REGION Network 2: Drive control B nok
   RUNG wire#powerrail
      Contact( "Servo Control"."B"."drive error" )
      wire#w1
      Coil( "Faults&warnings"."Status Nok"."Drive controller B NK" )
   END_RUNG
   RUNG wire#powerrail
      Contact( "Servo Control"."B"."Communication Error" )
   END_RUNG wire#w1
   RUNG wire#powerrail
      I_Contact( "Alarm Drive 2" )
   END_RUNG wire#w1
   RUNG wire#w1
      Coil( "Alarm_DB".input.alarm[10] )
   END_RUNG
   // the same network as SCL:
   "Faults&warnings"."Status Nok"."Drive controller B NK" := "Servo Control"."B"."drive error" OR "Servo Control"."B"."Communication Error" OR NOT "Alarm Drive 2";
   "Alarm_DB".input.alarm[10] := "Faults&warnings"."Status Nok"."Drive controller B NK";
END_REGION

REGION Network 3: Agitator A Fault
   RUNG wire#powerrail
      Contact( "A4-Agitator A1 fault" )
      Coil( "Faults&warnings"."Status Nok"."Agitator A Fault" )
   END_RUNG
   // the same network as SCL:
   "Faults&warnings"."Status Nok"."Agitator A Fault" := "A4-Agitator A1 fault";
END_REGION

REGION Network 4: Agitator B Fault
   RUNG wire#powerrail
      Contact( "A5-Agitator A2 fault" )
      Coil( "Faults&warnings"."Status Nok"."Agitator B Fault" )
   END_RUNG
   // the same network as SCL:
   "Faults&warnings"."Status Nok"."Agitator B Fault" := "A5-Agitator A2 fault";
END_REGION

REGION Network 5: pressure sensor Pump A inlet
   RUNG wire#powerrail
      { S7_Templates := "SrcType := Int" } GE_Contact(in1 := "Pressure sensor Pump Inlet A", in2 := 32767)
      { S7_Templates := "SrcType := Int" } EQ_Contact(in1 := "Control".Pressure_sensor_select, in2 := 0)
      wire#w1
      Coil( "Faults&warnings"."Status Nok"."Pressure sensor Pump A Inlet" )
   END_RUNG
   RUNG wire#powerrail
      { S7_Templates := "SrcType := Int" } GE_Contact(in1 := "Pressure sensor Pump Inlet A_mA", in2 := 32767)
      { S7_Templates := "SrcType := Int" } EQ_Contact(in1 := "Control".Pressure_sensor_select, in2 := 1)
   END_RUNG wire#w1
   // the same network as SCL:
   "Faults&warnings"."Status Nok"."Pressure sensor Pump A Inlet" := (("Pressure sensor Pump Inlet A" >= 32767) AND ("Control".Pressure_sensor_select = 0)) OR (("Pressure sensor Pump Inlet A_mA" >= 32767) AND ("Control".Pressure_sensor_select = 1));
END_REGION

REGION Network 6: pressure sensor Pump A outlet
   RUNG wire#powerrail
      { S7_Templates := "SrcType := Int" } GE_Contact(in1 := "Pressure Sensor Pump Outlet A", in2 := 32767)
      I_Contact( "AlwaysFALSE" )
      Contact( "pressure".Outlet_PT_ENABLE )
      wire#w1
      Coil( "Faults&warnings"."Status Nok"."Pressure sensor Pump A Outlet" )
   END_RUNG
   RUNG wire#w1
      Coil( "Alarm_DB".input.alarm[81] )
   END_RUNG
   // the same network as SCL:
   "Faults&warnings"."Status Nok"."Pressure sensor Pump A Outlet" := ("Pressure Sensor Pump Outlet A" >= 32767) AND NOT "AlwaysFALSE" AND "pressure".Outlet_PT_ENABLE;
   "Alarm_DB".input.alarm[81] := "Faults&warnings"."Status Nok"."Pressure sensor Pump A Outlet";
END_REGION

REGION Network 7: pressure sensor Pump B inlet
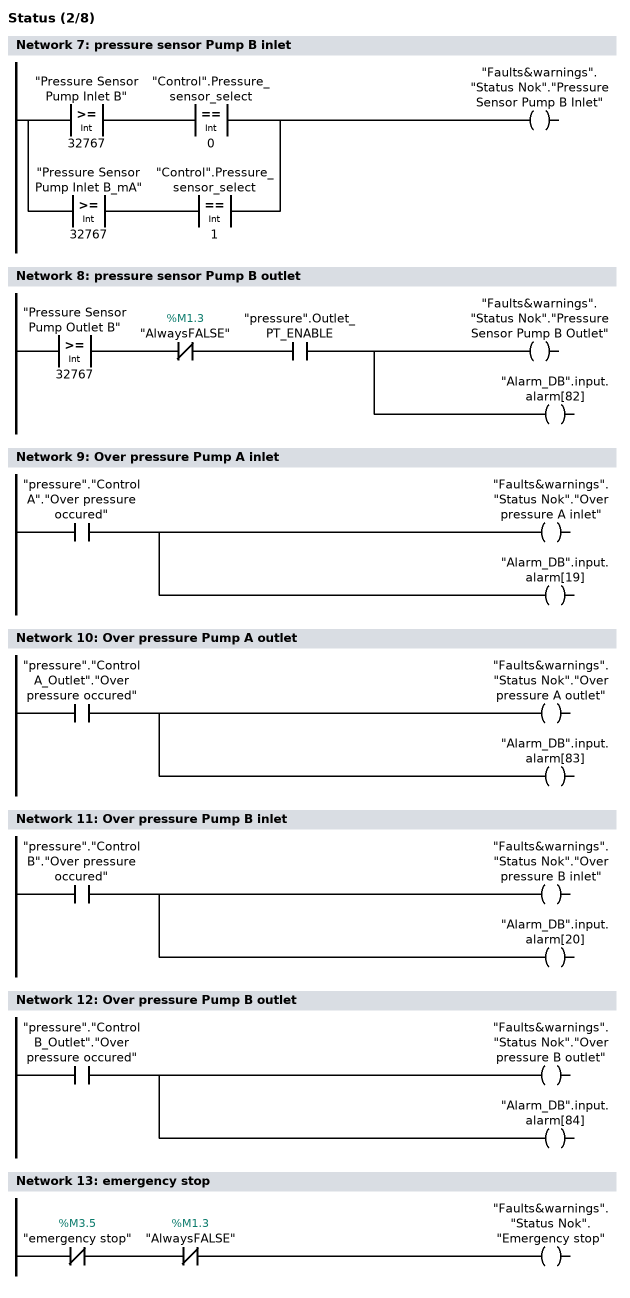
   RUNG wire#powerrail
      { S7_Templates := "SrcType := Int" } GE_Contact(in1 := "Pressure Sensor Pump Inlet B", in2 := 32767)
      { S7_Templates := "SrcType := Int" } EQ_Contact(in1 := "Control".Pressure_sensor_select, in2 := 0)
      wire#w1
      Coil( "Faults&warnings"."Status Nok"."Pressure Sensor Pump B Inlet" )
   END_RUNG
   RUNG wire#powerrail
      { S7_Templates := "SrcType := Int" } GE_Contact(in1 := "Pressure Sensor Pump Inlet B_mA", in2 := 32767)
      { S7_Templates := "SrcType := Int" } EQ_Contact(in1 := "Control".Pressure_sensor_select, in2 := 1)
   END_RUNG wire#w1
   // the same network as SCL:
   "Faults&warnings"."Status Nok"."Pressure Sensor Pump B Inlet" := (("Pressure Sensor Pump Inlet B" >= 32767) AND ("Control".Pressure_sensor_select = 0)) OR (("Pressure Sensor Pump Inlet B_mA" >= 32767) AND ("Control".Pressure_sensor_select = 1));
END_REGION

REGION Network 8: pressure sensor Pump B outlet
   RUNG wire#powerrail
      { S7_Templates := "SrcType := Int" } GE_Contact(in1 := "Pressure Sensor Pump Outlet B", in2 := 32767)
      I_Contact( "AlwaysFALSE" )
      Contact( "pressure".Outlet_PT_ENABLE )
      wire#w1
      Coil( "Faults&warnings"."Status Nok"."Pressure Sensor Pump B Outlet" )
   END_RUNG
   RUNG wire#w1
      Coil( "Alarm_DB".input.alarm[82] )
   END_RUNG
   // the same network as SCL:
   "Faults&warnings"."Status Nok"."Pressure Sensor Pump B Outlet" := ("Pressure Sensor Pump Outlet B" >= 32767) AND NOT "AlwaysFALSE" AND "pressure".Outlet_PT_ENABLE;
   "Alarm_DB".input.alarm[82] := "Faults&warnings"."Status Nok"."Pressure Sensor Pump B Outlet";
END_REGION

REGION Network 9: Over pressure Pump A inlet
   RUNG wire#powerrail
      Contact( "pressure"."Control A"."Over pressure occured" )
      wire#w1
      Coil( "Faults&warnings"."Status Nok"."Over pressure A inlet" )
   END_RUNG
   RUNG wire#w1
      Coil( "Alarm_DB".input.alarm[19] )
   END_RUNG
   // the same network as SCL:
   "Faults&warnings"."Status Nok"."Over pressure A inlet" := "pressure"."Control A"."Over pressure occured";
   "Alarm_DB".input.alarm[19] := "pressure"."Control A"."Over pressure occured";
END_REGION

REGION Network 10: Over pressure Pump A outlet
   RUNG wire#powerrail
      Contact( "pressure"."Control A_Outlet"."Over pressure occured" )
      wire#w1
      Coil( "Faults&warnings"."Status Nok"."Over pressure A outlet" )
   END_RUNG
   RUNG wire#w1
      Coil( "Alarm_DB".input.alarm[83] )
   END_RUNG
   // the same network as SCL:
   "Faults&warnings"."Status Nok"."Over pressure A outlet" := "pressure"."Control A_Outlet"."Over pressure occured";
   "Alarm_DB".input.alarm[83] := "pressure"."Control A_Outlet"."Over pressure occured";
END_REGION

REGION Network 11: Over pressure Pump B inlet
   RUNG wire#powerrail
      Contact( "pressure"."Control B"."Over pressure occured" )
      wire#w1
      Coil( "Faults&warnings"."Status Nok"."Over pressure B inlet" )
   END_RUNG
   RUNG wire#w1
      Coil( "Alarm_DB".input.alarm[20] )
   END_RUNG
   // the same network as SCL:
   "Faults&warnings"."Status Nok"."Over pressure B inlet" := "pressure"."Control B"."Over pressure occured";
   "Alarm_DB".input.alarm[20] := "pressure"."Control B"."Over pressure occured";
END_REGION

REGION Network 12: Over pressure Pump B outlet
   RUNG wire#powerrail
      Contact( "pressure"."Control B_Outlet"."Over pressure occured" )
      wire#w1
      Coil( "Faults&warnings"."Status Nok"."Over pressure B outlet" )
   END_RUNG
   RUNG wire#w1
      Coil( "Alarm_DB".input.alarm[84] )
   END_RUNG
   // the same network as SCL:
   "Faults&warnings"."Status Nok"."Over pressure B outlet" := "pressure"."Control B_Outlet"."Over pressure occured";
   "Alarm_DB".input.alarm[84] := "pressure"."Control B_Outlet"."Over pressure occured";
END_REGION

REGION Network 13: emergency stop
   RUNG wire#powerrail
      I_Contact( "emergency stop" )
      I_Contact( "AlwaysFALSE" )
      Coil( "Faults&warnings"."Status Nok"."Emergency stop" )
   END_RUNG
   // the same network as SCL:
   "Faults&warnings"."Status Nok"."Emergency stop" := NOT "emergency stop" AND NOT "AlwaysFALSE";
END_REGION

REGION Network 14: HEATER OK
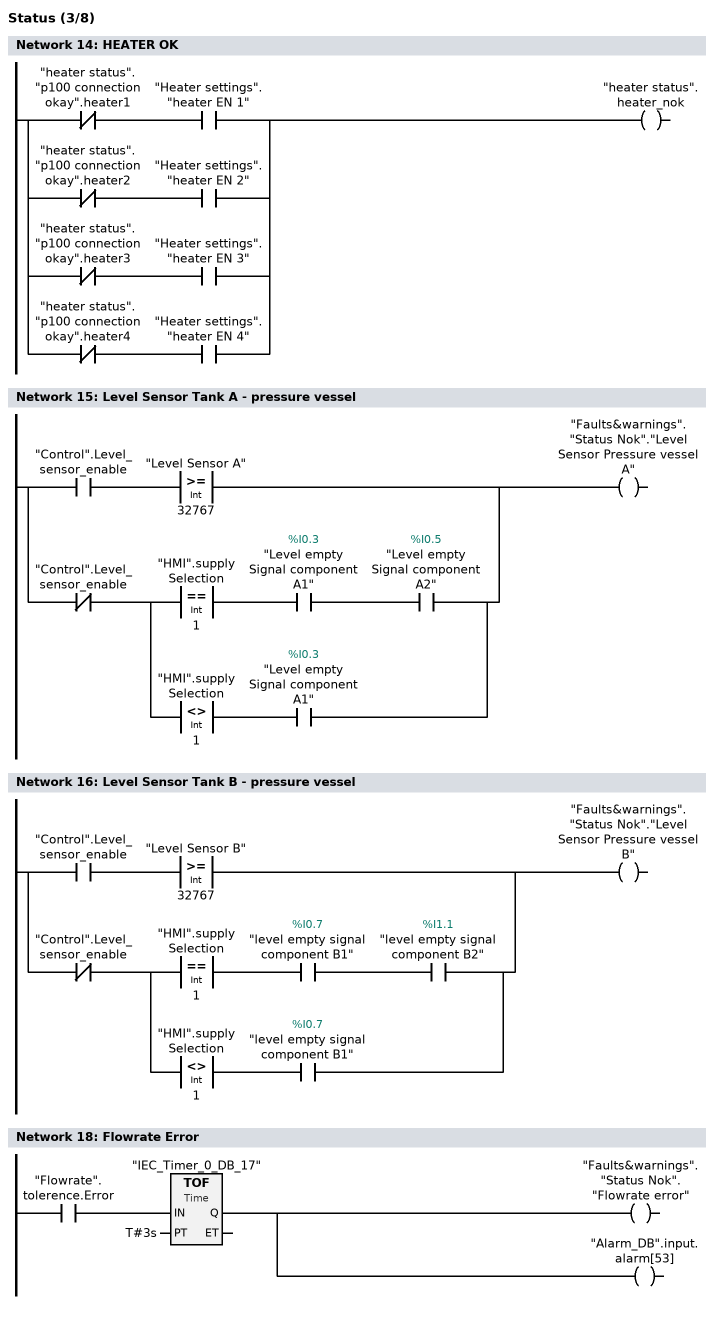
   RUNG wire#powerrail
      I_Contact( "heater status"."p100 connection okay".heater1 )
      Contact( "Heater settings"."heater EN 1" )
      wire#w1
      Coil( "heater status".heater_nok )
   END_RUNG
   RUNG wire#powerrail
      I_Contact( "heater status"."p100 connection okay".heater2 )
      Contact( "Heater settings"."heater EN 2" )
   END_RUNG wire#w1
   RUNG wire#powerrail
      I_Contact( "heater status"."p100 connection okay".heater3 )
      Contact( "Heater settings"."heater EN 3" )
   END_RUNG wire#w1
   RUNG wire#powerrail
      I_Contact( "heater status"."p100 connection okay".heater4 )
      Contact( "Heater settings"."heater EN 4" )
   END_RUNG wire#w1
   // the same network as SCL:
   "heater status".heater_nok := (NOT "heater status"."p100 connection okay".heater1 AND "Heater settings"."heater EN 1") OR (NOT "heater status"."p100 connection okay".heater2 AND "Heater settings"."heater EN 2") OR (NOT "heater status"."p100 connection okay".heater3 AND "Heater settings"."heater EN 3") OR (NOT "heater status"."p100 connection okay".heater4 AND "Heater settings"."heater EN 4");
END_REGION

REGION Network 15: Level Sensor Tank A - pressure vessel
   RUNG wire#powerrail
      Contact( "Control".Level_sensor_enable )
      { S7_Templates := "SrcType := Int" } GE_Contact(in1 := "Level Sensor A", in2 := 32767)
      wire#w1
      Coil( "Faults&warnings"."Status Nok"."Level Sensor Pressure vessel A" )
   END_RUNG
   RUNG wire#powerrail
      I_Contact( "Control".Level_sensor_enable )
      wire#w2
      { S7_Templates := "SrcType := Int" } EQ_Contact(in1 := "HMI".supplySelection, in2 := 1)
      Contact( "Level empty Signal component A1" )
      Contact( "Level empty Signal component A2" )
   END_RUNG wire#w1
   RUNG wire#w2
      { S7_Templates := "SrcType := Int" } NE_Contact(in1 := "HMI".supplySelection, in2 := 1)
      Contact( "Level empty Signal component A1" )
   END_RUNG wire#w1
   // the same network as SCL:
   "Faults&warnings"."Status Nok"."Level Sensor Pressure vessel A" := ("Control".Level_sensor_enable AND ("Level Sensor A" >= 32767)) OR (NOT "Control".Level_sensor_enable AND ((("HMI".supplySelection = 1) AND "Level empty Signal component A1" AND "Level empty Signal component A2") OR (("HMI".supplySelection <> 1) AND "Level empty Signal component A1")));
END_REGION

REGION Network 16: Level Sensor Tank B - pressure vessel
   RUNG wire#powerrail
      Contact( "Control".Level_sensor_enable )
      { S7_Templates := "SrcType := Int" } GE_Contact(in1 := "Level Sensor B", in2 := 32767)
      wire#w1
      Coil( "Faults&warnings"."Status Nok"."Level Sensor Pressure vessel B" )
   END_RUNG
   RUNG wire#powerrail
      I_Contact( "Control".Level_sensor_enable )
      wire#w2
      { S7_Templates := "SrcType := Int" } EQ_Contact(in1 := "HMI".supplySelection, in2 := 1)
      Contact( "level empty signal component B1" )
      Contact( "level empty signal component B2" )
   END_RUNG wire#w1
   RUNG wire#w2
      { S7_Templates := "SrcType := Int" } NE_Contact(in1 := "HMI".supplySelection, in2 := 1)
      Contact( "level empty signal component B1" )
   END_RUNG wire#w1
   // the same network as SCL:
   "Faults&warnings"."Status Nok"."Level Sensor Pressure vessel B" := ("Control".Level_sensor_enable AND ("Level Sensor B" >= 32767)) OR (NOT "Control".Level_sensor_enable AND ((("HMI".supplySelection = 1) AND "level empty signal component B1" AND "level empty signal component B2") OR (("HMI".supplySelection <> 1) AND "level empty signal component B1")));
END_REGION

REGION Network 17 (SCL): low level and empty level non tandum
   "Alarm_DB".input.alarm[40] := "Faults&warnings"."Status Nok"."Low level A1"  := "level"."Low level occured A";
   "Alarm_DB".input.alarm[42] := "Faults&warnings"."Status Nok"."Low level B1" := "level"."Low level occured B";

   "Faults&warnings"."Status Nok"."Level empty A1" := "level"."Level Empty A";
   "Alarm_DB".input.alarm[21] := "Faults&warnings"."Status Nok"."Level empty A1" OR "Temp".bit20;
   "Faults&warnings"."Status Nok"."Level empty B1" := "level"."Level Empty B";
   "Alarm_DB".input.alarm[23] := "Faults&warnings"."Status Nok"."Level empty B1" OR "Temp".bit21;

   "Faults&warnings"."Status Nok"."Level Low Drum A1" := "level"."Drum Level Low A1" AND "HMI".supplySelection = 1;
   "Faults&warnings"."Status Nok"."Level Low Drum A2" := "level"."Drum Level Low A2" AND "HMI".supplySelection = 1;
   "Faults&warnings"."Status Nok"."Level Low Drum B1" := "level"."Drum Level Low B1" AND "HMI".supplySelection = 1;
   "Faults&warnings"."Status Nok"."Level Low Drum B2" := "level"."Drum Level Low B2" AND "HMI".supplySelection = 1;

   "Faults&warnings"."Status Nok"."Level Empty Drum A1" := "level"."Drum Level Empty A1" AND "HMI".supplySelection = 1;
   "Faults&warnings"."Status Nok"."Level Empty Drum A2" := "level"."Drum Level Empty A2" AND "HMI".supplySelection = 1;
   "Faults&warnings"."Status Nok"."Level Empty Drum B1" := "level"."Drum Level Empty B1" AND "HMI".supplySelection = 1;
   "Faults&warnings"."Status Nok"."Level Empty Drum B2" := "level"."Drum Level Empty B2" AND "HMI".supplySelection = 1;
END_REGION

REGION Network 18: Flowrate Error
   RUNG wire#powerrail
      Contact( "Flowrate".tolerence.Error )
      { S7_Templates := "time_type := Time" } "IEC_Timer_0_DB_17".TOF(pt := T#3s, et =>)
      wire#w1
      Coil( "Faults&warnings"."Status Nok"."Flowrate error" )
   END_RUNG
   RUNG wire#w1
      Coil( "Alarm_DB".input.alarm[53] )
   END_RUNG
   // the same network as SCL:
   "IEC_Timer_0_DB_17".TOF(IN := "Flowrate".tolerence.Error, PT := T#3s);
   "Faults&warnings"."Status Nok"."Flowrate error" := "IEC_Timer_0_DB_17".Q;
   "Alarm_DB".input.alarm[53] := "IEC_Timer_0_DB_17".Q;
END_REGION

REGION Network 19: Critical Fault stop A metering
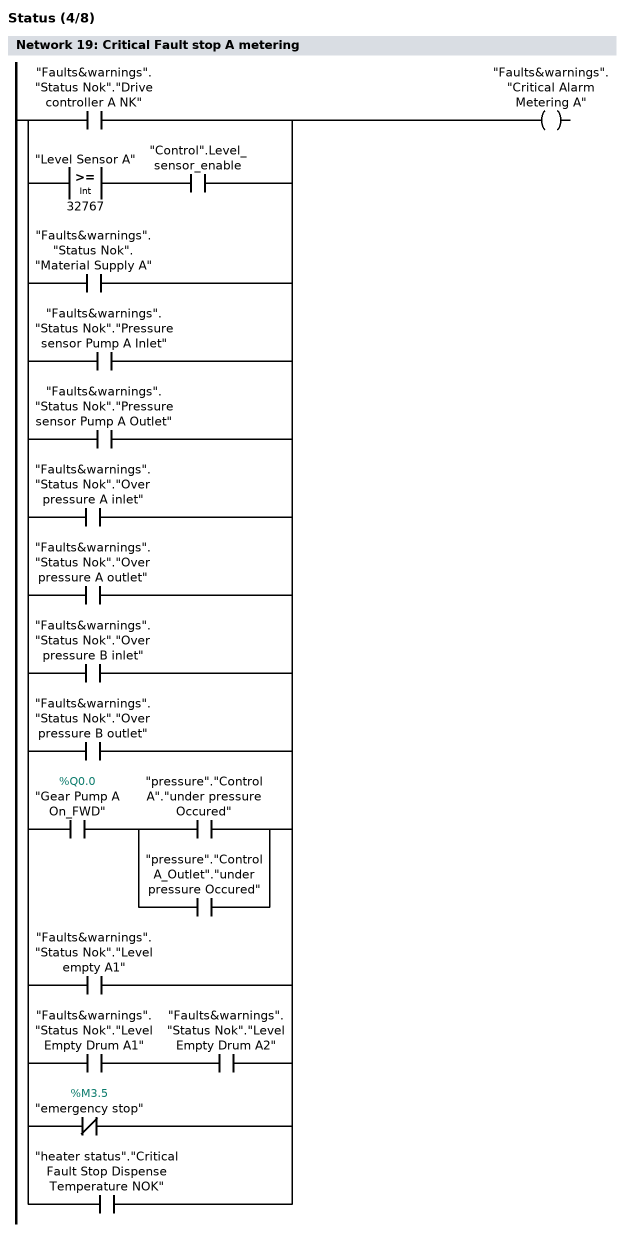
   RUNG wire#powerrail
      Contact( "Faults&warnings"."Status Nok"."Drive controller A NK" )
      wire#w1
      Coil( "Faults&warnings"."Critical Alarm Metering A" )
   END_RUNG
   RUNG wire#powerrail
      { S7_Templates := "SrcType := Int" } GE_Contact(in1 := "Level Sensor A", in2 := 32767)
      Contact( "Control".Level_sensor_enable )
   END_RUNG wire#w1
   RUNG wire#powerrail
      Contact( "Faults&warnings"."Status Nok"."Material Supply A" )
   END_RUNG wire#w1
   RUNG wire#powerrail
      Contact( "Faults&warnings"."Status Nok"."Pressure sensor Pump A Inlet" )
   END_RUNG wire#w1
   RUNG wire#powerrail
      Contact( "Faults&warnings"."Status Nok"."Pressure sensor Pump A Outlet" )
   END_RUNG wire#w1
   RUNG wire#powerrail
      Contact( "Faults&warnings"."Status Nok"."Over pressure A inlet" )
   END_RUNG wire#w1
   RUNG wire#powerrail
      Contact( "Faults&warnings"."Status Nok"."Over pressure A outlet" )
   END_RUNG wire#w1
   RUNG wire#powerrail
      Contact( "Faults&warnings"."Status Nok"."Over pressure B inlet" )
   END_RUNG wire#w1
   RUNG wire#powerrail
      Contact( "Faults&warnings"."Status Nok"."Over pressure B outlet" )
   END_RUNG wire#w1
   RUNG wire#powerrail
      Contact( "Gear Pump A On_FWD" )
      wire#w2
      Contact( "pressure"."Control A"."under pressure Occured" )
   END_RUNG wire#w1
   RUNG wire#w2
      Contact( "pressure"."Control A_Outlet"."under pressure Occured" )
   END_RUNG wire#w1
   RUNG wire#powerrail
      Contact( "Faults&warnings"."Status Nok"."Level empty A1" )
   END_RUNG wire#w1
   RUNG wire#powerrail
      Contact( "Faults&warnings"."Status Nok"."Level Empty Drum A1" )
      Contact( "Faults&warnings"."Status Nok"."Level Empty Drum A2" )
   END_RUNG wire#w1
   RUNG wire#powerrail
      I_Contact( "emergency stop" )
   END_RUNG wire#w1
   RUNG wire#powerrail
      Contact( "heater status"."Critical Fault Stop Dispense Temperature NOK" )
   END_RUNG wire#w1
   // the same network as SCL:
   "Faults&warnings"."Critical Alarm Metering A" := "Faults&warnings"."Status Nok"."Drive controller A NK" OR (("Level Sensor A" >= 32767) AND "Control".Level_sensor_enable) OR "Faults&warnings"."Status Nok"."Material Supply A" OR "Faults&warnings"."Status Nok"."Pressure sensor Pump A Inlet" OR "Faults&warnings"."Status Nok"."Pressure sensor Pump A Outlet" OR "Faults&warnings"."Status Nok"."Over pressure A inlet" OR "Faults&warnings"."Status Nok"."Over pressure A outlet" OR "Faults&warnings"."Status Nok"."Over pressure B inlet" OR "Faults&warnings"."Status Nok"."Over pressure B outlet" OR ("Gear Pump A On_FWD" AND ("pressure"."Control A"."under pressure Occured" OR "pressure"."Control A_Outlet"."under pressure Occured")) OR "Faults&warnings"."Status Nok"."Level empty A1" OR ("Faults&warnings"."Status Nok"."Level Empty Drum A1" AND "Faults&warnings"."Status Nok"."Level Empty Drum A2") OR NOT "emergency stop" OR "heater status"."Critical Fault Stop Dispense Temperature NOK";
END_REGION

REGION Network 20: Critical Fault stop B metering
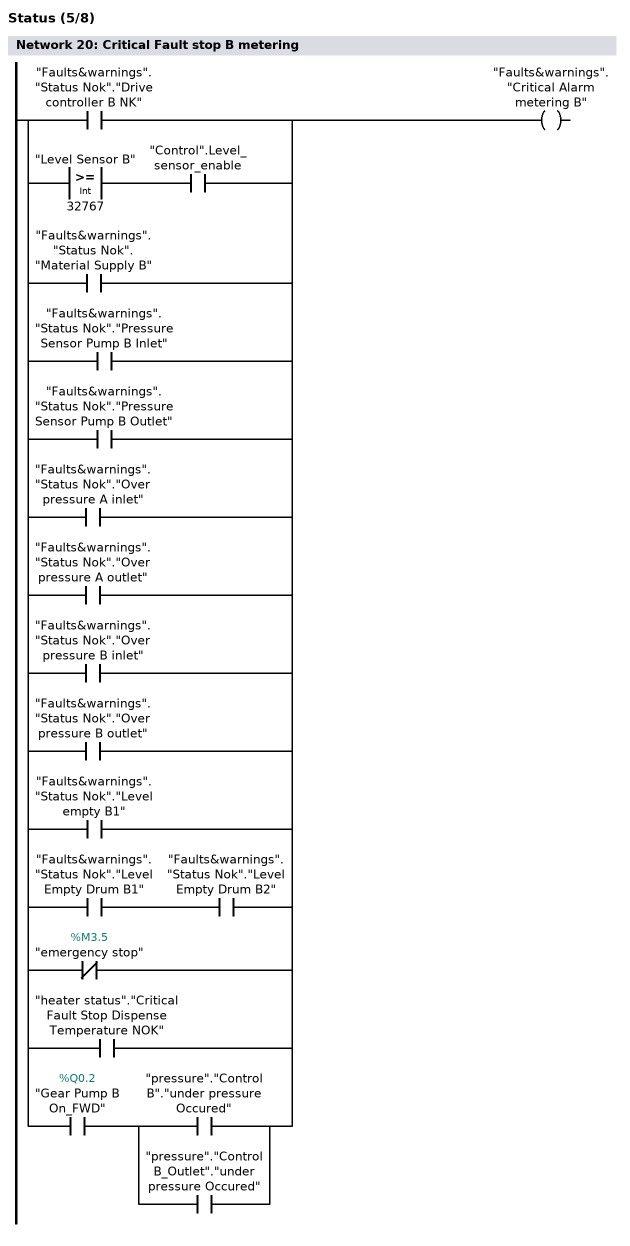
   RUNG wire#powerrail
      Contact( "Faults&warnings"."Status Nok"."Drive controller B NK" )
      wire#w1
      Coil( "Faults&warnings"."Critical Alarm metering B" )
   END_RUNG
   RUNG wire#powerrail
      { S7_Templates := "SrcType := Int" } GE_Contact(in1 := "Level Sensor B", in2 := 32767)
      Contact( "Control".Level_sensor_enable )
   END_RUNG wire#w1
   RUNG wire#powerrail
      Contact( "Faults&warnings"."Status Nok"."Material Supply B" )
   END_RUNG wire#w1
   RUNG wire#powerrail
      Contact( "Faults&warnings"."Status Nok"."Pressure Sensor Pump B Inlet" )
   END_RUNG wire#w1
   RUNG wire#powerrail
      Contact( "Faults&warnings"."Status Nok"."Pressure Sensor Pump B Outlet" )
   END_RUNG wire#w1
   RUNG wire#powerrail
      Contact( "Faults&warnings"."Status Nok"."Over pressure A inlet" )
   END_RUNG wire#w1
   RUNG wire#powerrail
      Contact( "Faults&warnings"."Status Nok"."Over pressure A outlet" )
   END_RUNG wire#w1
   RUNG wire#powerrail
      Contact( "Faults&warnings"."Status Nok"."Over pressure B inlet" )
   END_RUNG wire#w1
   RUNG wire#powerrail
      Contact( "Faults&warnings"."Status Nok"."Over pressure B outlet" )
   END_RUNG wire#w1
   RUNG wire#powerrail
      Contact( "Faults&warnings"."Status Nok"."Level empty B1" )
   END_RUNG wire#w1
   RUNG wire#powerrail
      Contact( "Faults&warnings"."Status Nok"."Level Empty Drum B1" )
      Contact( "Faults&warnings"."Status Nok"."Level Empty Drum B2" )
   END_RUNG wire#w1
   RUNG wire#powerrail
      I_Contact( "emergency stop" )
   END_RUNG wire#w1
   RUNG wire#powerrail
      Contact( "heater status"."Critical Fault Stop Dispense Temperature NOK" )
   END_RUNG wire#w1
   RUNG wire#powerrail
      Contact( "Gear Pump B On_FWD" )
      wire#w2
      Contact( "pressure"."Control B"."under pressure Occured" )
   END_RUNG wire#w1
   RUNG wire#w2
      Contact( "pressure"."Control B_Outlet"."under pressure Occured" )
   END_RUNG wire#w1
   // the same network as SCL:
   "Faults&warnings"."Critical Alarm metering B" := "Faults&warnings"."Status Nok"."Drive controller B NK" OR (("Level Sensor B" >= 32767) AND "Control".Level_sensor_enable) OR "Faults&warnings"."Status Nok"."Material Supply B" OR "Faults&warnings"."Status Nok"."Pressure Sensor Pump B Inlet" OR "Faults&warnings"."Status Nok"."Pressure Sensor Pump B Outlet" OR "Faults&warnings"."Status Nok"."Over pressure A inlet" OR "Faults&warnings"."Status Nok"."Over pressure A outlet" OR "Faults&warnings"."Status Nok"."Over pressure B inlet" OR "Faults&warnings"."Status Nok"."Over pressure B outlet" OR "Faults&warnings"."Status Nok"."Level empty B1" OR ("Faults&warnings"."Status Nok"."Level Empty Drum B1" AND "Faults&warnings"."Status Nok"."Level Empty Drum B2") OR NOT "emergency stop" OR "heater status"."Critical Fault Stop Dispense Temperature NOK" OR ("Gear Pump B On_FWD" AND ("pressure"."Control B"."under pressure Occured" OR "pressure"."Control B_Outlet"."under pressure Occured"));
END_REGION

REGION Network 21: critical alarm AB
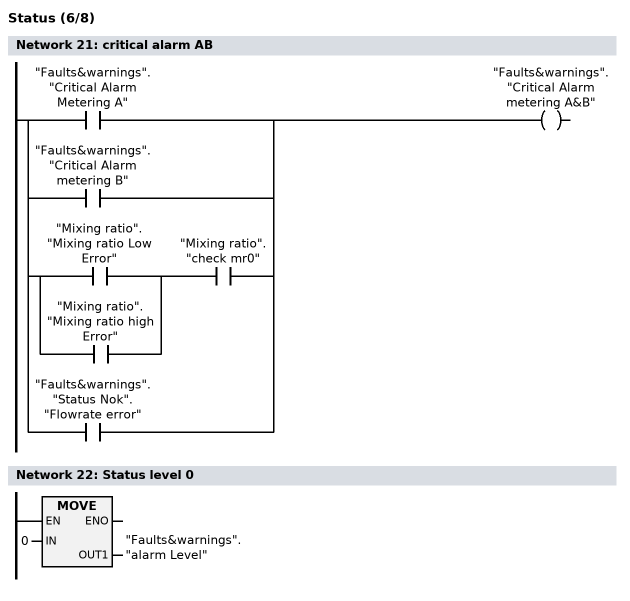
   RUNG wire#powerrail
      Contact( "Faults&warnings"."Critical Alarm Metering A" )
      wire#w1
      Coil( "Faults&warnings"."Critical Alarm metering A&B" )
   END_RUNG
   RUNG wire#powerrail
      Contact( "Faults&warnings"."Critical Alarm metering B" )
   END_RUNG wire#w1
   RUNG wire#powerrail
      Contact( "Mixing ratio"."Mixing ratio Low  Error" )
      wire#w2
      Contact( "Mixing ratio"."check mr0" )
   END_RUNG wire#w1
   RUNG wire#powerrail
      Contact( "Mixing ratio"."Mixing ratio high Error" )
   END_RUNG wire#w2
   RUNG wire#powerrail
      Contact( "Faults&warnings"."Status Nok"."Flowrate error" )
   END_RUNG wire#w1
   // the same network as SCL:
   "Faults&warnings"."Critical Alarm metering A&B" := "Faults&warnings"."Critical Alarm Metering A" OR "Faults&warnings"."Critical Alarm metering B" OR (("Mixing ratio"."Mixing ratio Low  Error" OR "Mixing ratio"."Mixing ratio high Error") AND "Mixing ratio"."check mr0") OR "Faults&warnings"."Status Nok"."Flowrate error";
END_REGION

REGION Network 22: Status level 0
   RUNG wire#powerrail
      Move(in := 0, out1 => "Faults&warnings"."alarm Level")
   END_RUNG
   // the same network as SCL:
   "Faults&warnings"."alarm Level" := 0;
END_REGION

REGION Network 23: Status level 1/warning
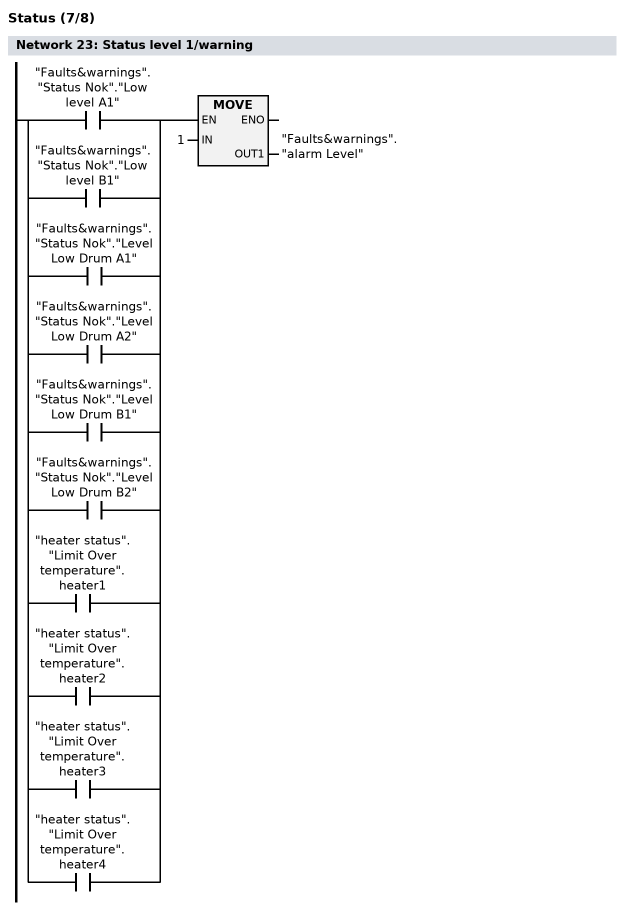
   RUNG wire#powerrail
      Contact( "Faults&warnings"."Status Nok"."Low level A1" )
      wire#w1
      Move(in := 1, out1 => "Faults&warnings"."alarm Level")
   END_RUNG
   RUNG wire#powerrail
      Contact( "Faults&warnings"."Status Nok"."Low level B1" )
   END_RUNG wire#w1
   RUNG wire#powerrail
      Contact( "Faults&warnings"."Status Nok"."Level Low Drum A1" )
   END_RUNG wire#w1
   RUNG wire#powerrail
      Contact( "Faults&warnings"."Status Nok"."Level Low Drum A2" )
   END_RUNG wire#w1
   RUNG wire#powerrail
      Contact( "Faults&warnings"."Status Nok"."Level Low Drum B1" )
   END_RUNG wire#w1
   RUNG wire#powerrail
      Contact( "Faults&warnings"."Status Nok"."Level Low Drum B2" )
   END_RUNG wire#w1
   RUNG wire#powerrail
      Contact( "heater status"."Limit Over temperature".heater1 )
   END_RUNG wire#w1
   RUNG wire#powerrail
      Contact( "heater status"."Limit Over temperature".heater2 )
   END_RUNG wire#w1
   RUNG wire#powerrail
      Contact( "heater status"."Limit Over temperature".heater3 )
   END_RUNG wire#w1
   RUNG wire#powerrail
      Contact( "heater status"."Limit Over temperature".heater4 )
   END_RUNG wire#w1
   // the same network as SCL:
   IF "Faults&warnings"."Status Nok"."Low level A1" OR "Faults&warnings"."Status Nok"."Low level B1" OR "Faults&warnings"."Status Nok"."Level Low Drum A1" OR "Faults&warnings"."Status Nok"."Level Low Drum A2" OR "Faults&warnings"."Status Nok"."Level Low Drum B1" OR "Faults&warnings"."Status Nok"."Level Low Drum B2" OR "heater status"."Limit Over temperature".heater1 OR "heater status"."Limit Over temperature".heater2 OR "heater status"."Limit Over temperature".heater3 OR "heater status"."Limit Over temperature".heater4 THEN
       "Faults&warnings"."alarm Level" := 1;
   END_IF;
END_REGION

REGION Network 24: Status level 1/fault
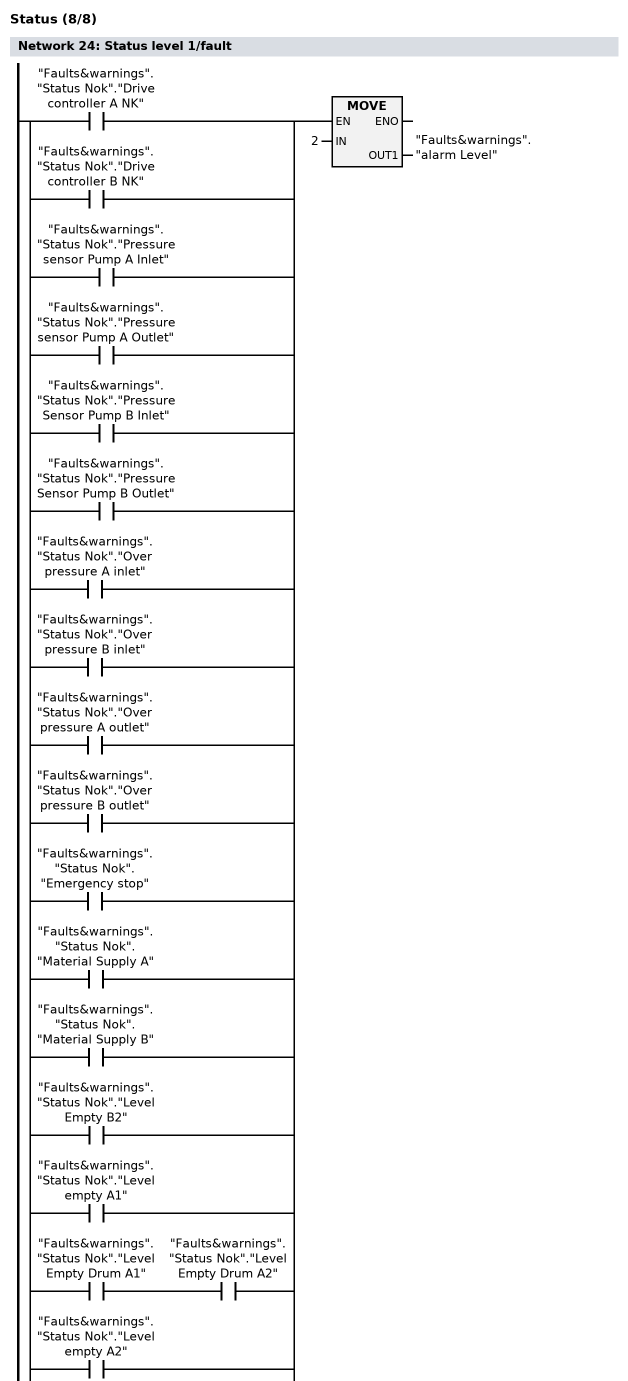
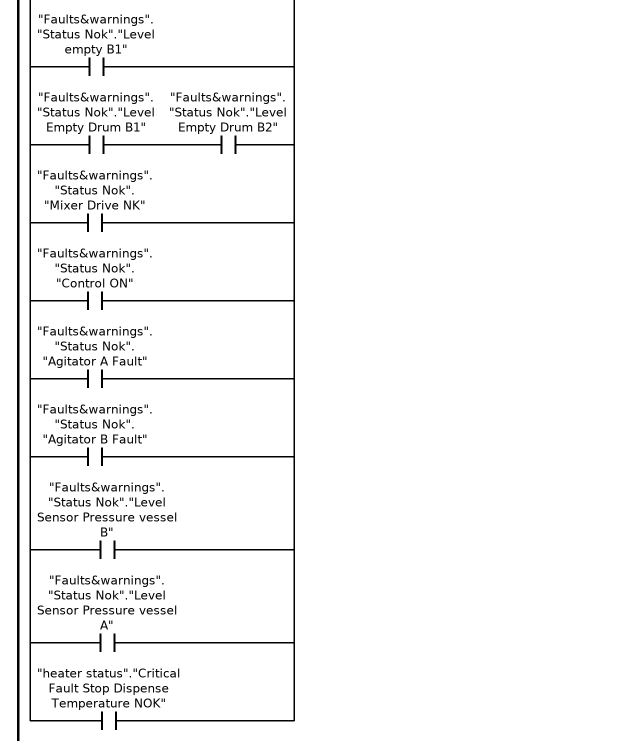
   RUNG wire#powerrail
      Contact( "Faults&warnings"."Status Nok"."Drive controller A NK" )
      wire#w1
      Move(in := 2, out1 => "Faults&warnings"."alarm Level")
   END_RUNG
   RUNG wire#powerrail
      Contact( "Faults&warnings"."Status Nok"."Drive controller B NK" )
   END_RUNG wire#w1
   RUNG wire#powerrail
      Contact( "Faults&warnings"."Status Nok"."Pressure sensor Pump A Inlet" )
   END_RUNG wire#w1
   RUNG wire#powerrail
      Contact( "Faults&warnings"."Status Nok"."Pressure sensor Pump A Outlet" )
   END_RUNG wire#w1
   RUNG wire#powerrail
      Contact( "Faults&warnings"."Status Nok"."Pressure Sensor Pump B Inlet" )
   END_RUNG wire#w1
   RUNG wire#powerrail
      Contact( "Faults&warnings"."Status Nok"."Pressure Sensor Pump B Outlet" )
   END_RUNG wire#w1
   RUNG wire#powerrail
      Contact( "Faults&warnings"."Status Nok"."Over pressure A inlet" )
   END_RUNG wire#w1
   RUNG wire#powerrail
      Contact( "Faults&warnings"."Status Nok"."Over pressure B inlet" )
   END_RUNG wire#w1
   RUNG wire#powerrail
      Contact( "Faults&warnings"."Status Nok"."Over pressure A outlet" )
   END_RUNG wire#w1
   RUNG wire#powerrail
      Contact( "Faults&warnings"."Status Nok"."Over pressure B outlet" )
   END_RUNG wire#w1
   RUNG wire#powerrail
      Contact( "Faults&warnings"."Status Nok"."Emergency stop" )
   END_RUNG wire#w1
   RUNG wire#powerrail
      Contact( "Faults&warnings"."Status Nok"."Material Supply A" )
   END_RUNG wire#w1
   RUNG wire#powerrail
      Contact( "Faults&warnings"."Status Nok"."Material Supply B" )
   END_RUNG wire#w1
   RUNG wire#powerrail
      Contact( "Faults&warnings"."Status Nok"."Level Empty B2" )
   END_RUNG wire#w1
   RUNG wire#powerrail
      Contact( "Faults&warnings"."Status Nok"."Level empty A1" )
   END_RUNG wire#w1
   RUNG wire#powerrail
      Contact( "Faults&warnings"."Status Nok"."Level Empty Drum A1" )
      Contact( "Faults&warnings"."Status Nok"."Level Empty Drum A2" )
   END_RUNG wire#w1
   RUNG wire#powerrail
      Contact( "Faults&warnings"."Status Nok"."Level empty A2" )
   END_RUNG wire#w1
   RUNG wire#powerrail
      Contact( "Faults&warnings"."Status Nok"."Level empty B1" )
   END_RUNG wire#w1
   RUNG wire#powerrail
      Contact( "Faults&warnings"."Status Nok"."Level Empty Drum B1" )
      Contact( "Faults&warnings"."Status Nok"."Level Empty Drum B2" )
   END_RUNG wire#w1
   RUNG wire#powerrail
      Contact( "Faults&warnings"."Status Nok"."Mixer Drive NK" )
   END_RUNG wire#w1
   RUNG wire#powerrail
      Contact( "Faults&warnings"."Status Nok"."Control ON" )
   END_RUNG wire#w1
   RUNG wire#powerrail
      Contact( "Faults&warnings"."Status Nok"."Agitator A Fault" )
   END_RUNG wire#w1
   RUNG wire#powerrail
      Contact( "Faults&warnings"."Status Nok"."Agitator B Fault" )
   END_RUNG wire#w1
   RUNG wire#powerrail
      Contact( "Faults&warnings"."Status Nok"."Level Sensor Pressure vessel B" )
   END_RUNG wire#w1
   RUNG wire#powerrail
      Contact( "Faults&warnings"."Status Nok"."Level Sensor Pressure vessel A" )
   END_RUNG wire#w1
   RUNG wire#powerrail
      Contact( "heater status"."Critical Fault Stop Dispense Temperature NOK" )
   END_RUNG wire#w1
   // the same network as SCL:
   IF "Faults&warnings"."Status Nok"."Drive controller A NK" OR "Faults&warnings"."Status Nok"."Drive controller B NK" OR "Faults&warnings"."Status Nok"."Pressure sensor Pump A Inlet" OR "Faults&warnings"."Status Nok"."Pressure sensor Pump A Outlet" OR "Faults&warnings"."Status Nok"."Pressure Sensor Pump B Inlet" OR "Faults&warnings"."Status Nok"."Pressure Sensor Pump B Outlet" OR "Faults&warnings"."Status Nok"."Over pressure A inlet" OR "Faults&warnings"."Status Nok"."Over pressure B inlet" OR "Faults&warnings"."Status Nok"."Over pressure A outlet" OR "Faults&warnings"."Status Nok"."Over pressure B outlet" OR "Faults&warnings"."Status Nok"."Emergency stop" OR "Faults&warnings"."Status Nok"."Material Supply A" OR "Faults&warnings"."Status Nok"."Material Supply B" OR "Faults&warnings"."Status Nok"."Level Empty B2" OR "Faults&warnings"."Status Nok"."Level empty A1" OR ("Faults&warnings"."Status Nok"."Level Empty Drum A1" AND "Faults&warnings"."Status Nok"."Level Empty Drum A2") OR "Faults&warnings"."Status Nok"."Level empty A2" OR "Faults&warnings"."Status Nok"."Level empty B1" OR ("Faults&warnings"."Status Nok"."Level Empty Drum B1" AND "Faults&warnings"."Status Nok"."Level Empty Drum B2") OR "Faults&warnings"."Status Nok"."Mixer Drive NK" OR "Faults&warnings"."Status Nok"."Control ON" OR "Faults&warnings"."Status Nok"."Agitator A Fault" OR "Faults&warnings"."Status Nok"."Agitator B Fault" OR "Faults&warnings"."Status Nok"."Level Sensor Pressure vessel B" OR "Faults&warnings"."Status Nok"."Level Sensor Pressure vessel A" OR "heater status"."Critical Fault Stop Dispense Temperature NOK" THEN
       "Faults&warnings"."alarm Level" := 2;
   END_IF;
END_REGION
END_FUNCTION

FUNCTION "Pressure control" : Void   // FC24, LAD
{ S7_Optimized_Access := 'TRUE' }
VERSION : 0.1
// stored: AutoNumber true, IsIECCheckEnabled false, SetENOAutomatically false, UDAEnableTagReadback false
BEGIN

REGION Network 1 (SCL): Pump A pressure setting Inlet

   IF "Pressure sensor Pump Inlet A" < 32767 AND "Control".Pressure_sensor_select = 0 THEN
       "pressure".Misc."Pump A Scalx valueIN" := SCALE_X(MIN := 0.0,
                                                           VALUE := NORM_X(MIN := 0,
                                                                           VALUE := "Pressure sensor Pump Inlet A",
                                                                           MAX := 27648),
                                                           MAX := "pressure".A."pressure at 20mA");
   ELSIF "Pressure sensor Pump Inlet A_mA" < 32767 AND "Control".Pressure_sensor_select = 1 THEN
       "pressure".Misc."Pump A Scalx valueIN" := SCALE_X(MIN := 0.0,
                                                           VALUE := NORM_X(MIN := 0,
                                                                           VALUE := "Pressure sensor Pump Inlet A_mA",
                                                                           MAX := 27648),
                                                           MAX := "pressure".A."pressure at 20mA");
   END_IF;

   "Alarm_DB".input.alarm[15] := (("Control".Pressure_sensor_select = 0) AND ("Pressure sensor Pump Inlet A" >= 32767)) OR (("Control".Pressure_sensor_select = 1) AND ("Pressure sensor Pump Inlet A_mA" >= 32767));
END_REGION

REGION Network 2 (SCL): Pump A pressure setting Outlet

   IF "Pressure Sensor Pump Outlet A" < 32767 THEN
       "pressure".Misc."Pump A Scalx valueOUT" := SCALE_X(MIN := 0.0,
                                                           VALUE := NORM_X(MIN := 0,
                                                                           VALUE := "Pressure Sensor Pump Outlet A",
                                                                           MAX := 27648),
                                                           MAX := "pressure".A_Outlet."pressure at 20mA");
   END_IF;
END_REGION

REGION Network 3: gear Pump A pressure
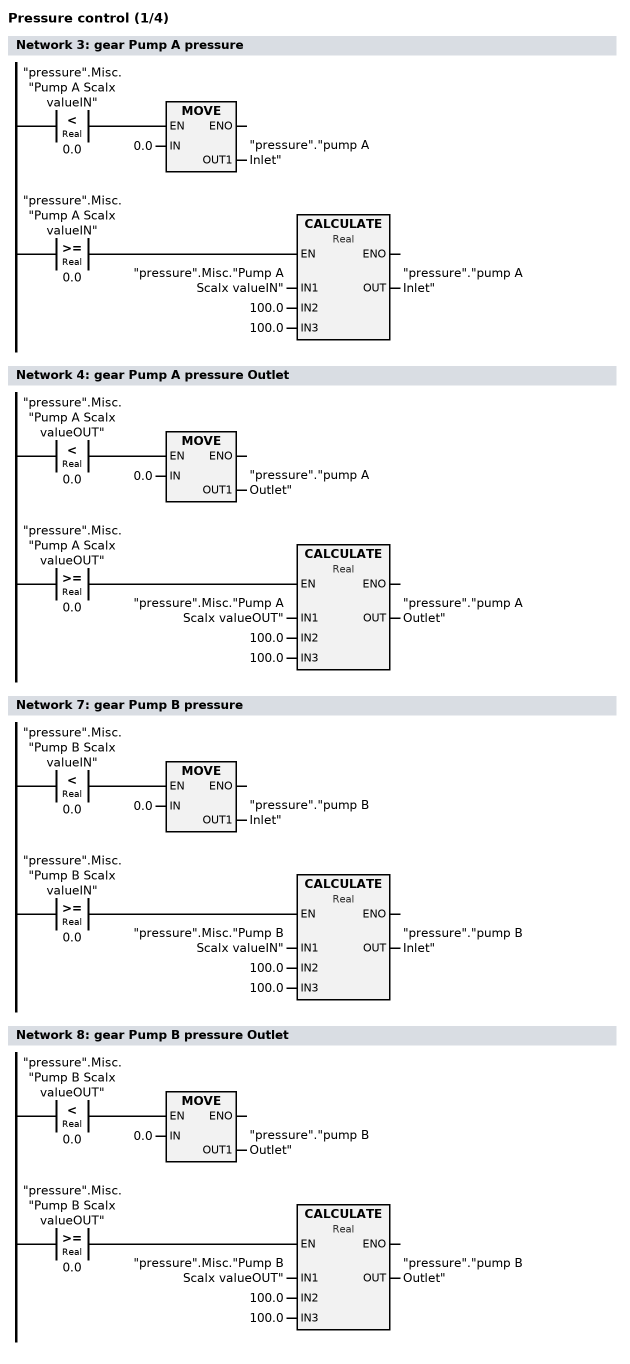
   RUNG wire#powerrail
      { S7_Templates := "SrcType := Real" } LT_Contact(in1 := "pressure".Misc."Pump A Scalx valueIN", in2 := 0.0)
      Move(in := 0.0, out1 => "pressure"."pump A Inlet")
   END_RUNG
   RUNG wire#powerrail
      { S7_Templates := "SrcType := Real" } GE_Contact(in1 := "pressure".Misc."Pump A Scalx valueIN", in2 := 0.0)
      { S7_Templates := "SrcType := Real"; S7_Expression := "ROUND(IN1*IN2)/IN3" } Calculate(in1 := "pressure".Misc."Pump A Scalx valueIN", in2 := 100.0, in3 := 100.0, out => "pressure"."pump A Inlet")
   END_RUNG
   // the same network as SCL:
   IF "pressure".Misc."Pump A Scalx valueIN" < 0.0 THEN "pressure"."pump A Inlet" := 0.0; END_IF;
   IF "pressure".Misc."Pump A Scalx valueIN" >= 0.0 THEN
       "pressure"."pump A Inlet" := ROUND("pressure".Misc."Pump A Scalx valueIN"*100.0)/100.0;
   END_IF;
END_REGION

REGION Network 4: gear Pump A pressure Outlet
   RUNG wire#powerrail
      { S7_Templates := "SrcType := Real" } LT_Contact(in1 := "pressure".Misc."Pump A Scalx valueOUT", in2 := 0.0)
      Move(in := 0.0, out1 => "pressure"."pump A Outlet")
   END_RUNG
   RUNG wire#powerrail
      { S7_Templates := "SrcType := Real" } GE_Contact(in1 := "pressure".Misc."Pump A Scalx valueOUT", in2 := 0.0)
      { S7_Templates := "SrcType := Real"; S7_Expression := "ROUND(IN1*IN2)/IN3" } Calculate(in1 := "pressure".Misc."Pump A Scalx valueOUT", in2 := 100.0, in3 := 100.0, out => "pressure"."pump A Outlet")
   END_RUNG
   // the same network as SCL:
   IF "pressure".Misc."Pump A Scalx valueOUT" < 0.0 THEN "pressure"."pump A Outlet" := 0.0; END_IF;
   IF "pressure".Misc."Pump A Scalx valueOUT" >= 0.0 THEN
       "pressure"."pump A Outlet" := ROUND("pressure".Misc."Pump A Scalx valueOUT"*100.0)/100.0;
   END_IF;
END_REGION

REGION Network 5 (SCL): Pump b pressure setting Inlet

   IF "Pressure Sensor Pump Inlet B" < 32767 AND "Control".Pressure_sensor_select = 0 THEN
       "pressure".Misc."Pump B Scalx valueIN" := SCALE_X(MIN := 0.0,
                                                           VALUE := NORM_X(MIN := 0,
                                                                           VALUE := "Pressure Sensor Pump Inlet B",
                                                                           MAX := 27648),
                                                           MAX := "pressure".B."pressure at 20mA");
   ELSIF "Pressure Sensor Pump Inlet B_mA" < 32767 AND "Control".Pressure_sensor_select = 1 THEN
       "pressure".Misc."Pump B Scalx valueIN" := SCALE_X(MIN := 0.0,
                                                           VALUE := NORM_X(MIN := 0,
                                                                           VALUE := "Pressure Sensor Pump Inlet B_mA",
                                                                           MAX := 27648),
                                                           MAX := "pressure".B."pressure at 20mA");
   END_IF;
   "Alarm_DB".input.alarm[0] := (("Control".Pressure_sensor_select = 0) AND ("Pressure Sensor Pump Inlet B" >= 32767)) OR (("Control".Pressure_sensor_select = 1) AND ("Pressure Sensor Pump Inlet B_mA" >= 32767));
END_REGION

REGION Network 6 (SCL): Pump b pressure setting Outlet

   IF "Pressure Sensor Pump Outlet B" < 32767 THEN
       "pressure".Misc."Pump B Scalx valueOUT" := SCALE_X(MIN := 0.0,
                                                           VALUE := NORM_X(MIN := 0,
                                                                           VALUE := "Pressure Sensor Pump Outlet B",
                                                                           MAX := 27648),
                                                           MAX := "pressure".B_Outlet."pressure at 20mA");
   END_IF;
END_REGION

REGION Network 7: gear Pump B pressure
   RUNG wire#powerrail
      { S7_Templates := "SrcType := Real" } LT_Contact(in1 := "pressure".Misc."Pump B Scalx valueIN", in2 := 0.0)
      Move(in := 0.0, out1 => "pressure"."pump B Inlet")
   END_RUNG
   RUNG wire#powerrail
      { S7_Templates := "SrcType := Real" } GE_Contact(in1 := "pressure".Misc."Pump B Scalx valueIN", in2 := 0.0)
      { S7_Templates := "SrcType := Real"; S7_Expression := "ROUND(IN1*IN2)/IN3" } Calculate(in1 := "pressure".Misc."Pump B Scalx valueIN", in2 := 100.0, in3 := 100.0, out => "pressure"."pump B Inlet")
   END_RUNG
   // the same network as SCL:
   IF "pressure".Misc."Pump B Scalx valueIN" < 0.0 THEN "pressure"."pump B Inlet" := 0.0; END_IF;
   IF "pressure".Misc."Pump B Scalx valueIN" >= 0.0 THEN
       "pressure"."pump B Inlet" := ROUND("pressure".Misc."Pump B Scalx valueIN"*100.0)/100.0;
   END_IF;
END_REGION

REGION Network 8: gear Pump B pressure Outlet
   RUNG wire#powerrail
      { S7_Templates := "SrcType := Real" } LT_Contact(in1 := "pressure".Misc."Pump B Scalx valueOUT", in2 := 0.0)
      Move(in := 0.0, out1 => "pressure"."pump B Outlet")
   END_RUNG
   RUNG wire#powerrail
      { S7_Templates := "SrcType := Real" } GE_Contact(in1 := "pressure".Misc."Pump B Scalx valueOUT", in2 := 0.0)
      { S7_Templates := "SrcType := Real"; S7_Expression := "ROUND(IN1*IN2)/IN3" } Calculate(in1 := "pressure".Misc."Pump B Scalx valueOUT", in2 := 100.0, in3 := 100.0, out => "pressure"."pump B Outlet")
   END_RUNG
   // the same network as SCL:
   IF "pressure".Misc."Pump B Scalx valueOUT" < 0.0 THEN "pressure"."pump B Outlet" := 0.0; END_IF;
   IF "pressure".Misc."Pump B Scalx valueOUT" >= 0.0 THEN
       "pressure"."pump B Outlet" := ROUND("pressure".Misc."Pump B Scalx valueOUT"*100.0)/100.0;
   END_IF;
END_REGION

REGION Network 9: mbar to bar
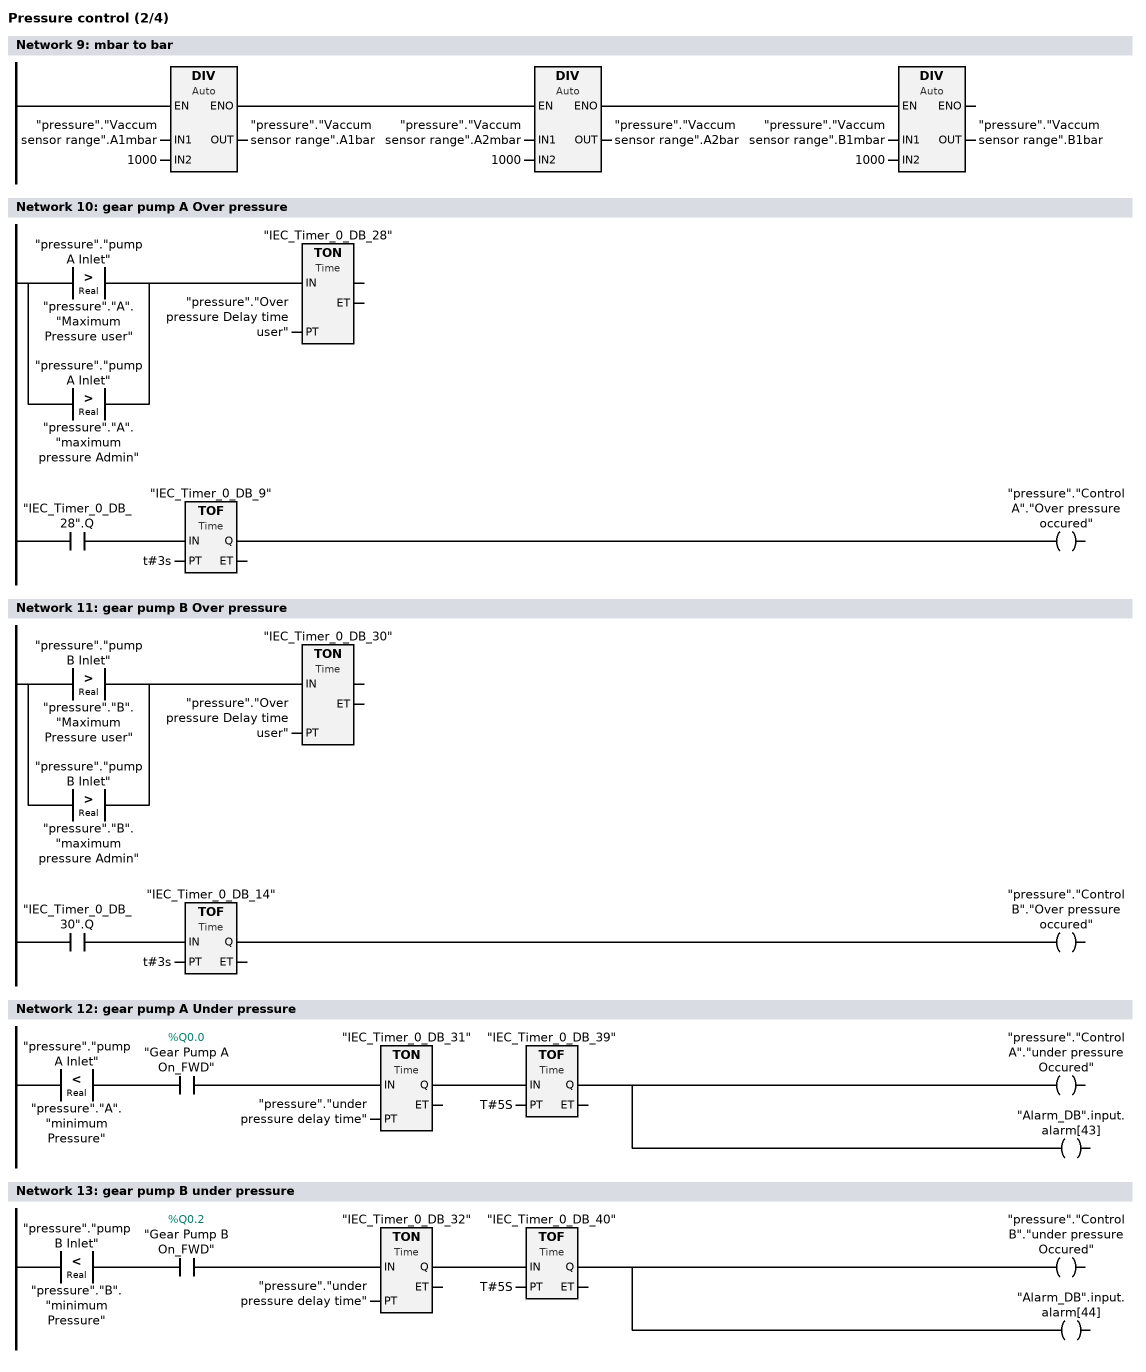
   RUNG wire#powerrail
      Div(in1 := "pressure"."Vaccum  sensor range".A1mbar, in2 := 1000, out => "pressure"."Vaccum  sensor range".A1bar)
      Div(in1 := "pressure"."Vaccum  sensor range".A2mbar, in2 := 1000, out => "pressure"."Vaccum  sensor range".A2bar)
      Div(in1 := "pressure"."Vaccum  sensor range".B1mbar, in2 := 1000, out => "pressure"."Vaccum  sensor range".B1bar)
   END_RUNG
   // the same network as SCL:
   "pressure"."Vaccum  sensor range".A1bar := "pressure"."Vaccum  sensor range".A1mbar / 1000;
   "pressure"."Vaccum  sensor range".A2bar := "pressure"."Vaccum  sensor range".A2mbar / 1000;
   "pressure"."Vaccum  sensor range".B1bar := "pressure"."Vaccum  sensor range".B1mbar / 1000;
END_REGION

REGION Network 10: gear pump A Over pressure
   RUNG wire#powerrail
      { S7_Templates := "SrcType := Real" } GT_Contact(in1 := "pressure"."pump A Inlet", in2 := "pressure"."A"."Maximum Pressure user")
      wire#w1
      { S7_Templates := "time_type := Time" } "IEC_Timer_0_DB_28".TON(pt := "pressure"."Over pressure Delay time user", et =>)
   END_RUNG
   RUNG wire#powerrail
      { S7_Templates := "SrcType := Real" } GT_Contact(in1 := "pressure"."pump A Inlet", in2 := "pressure"."A"."maximum pressure Admin")
   END_RUNG wire#w1
   RUNG wire#powerrail
      Contact( "IEC_Timer_0_DB_28".Q )
      { S7_Templates := "time_type := Time" } "IEC_Timer_0_DB_9".TOF(pt := t#3s, et =>)
      Coil( "pressure"."Control A"."Over pressure occured" )
   END_RUNG
   // the same network as SCL:
   "IEC_Timer_0_DB_28".TON(IN := ("pressure"."pump A Inlet" > "pressure"."A"."Maximum Pressure user") OR ("pressure"."pump A Inlet" > "pressure"."A"."maximum pressure Admin"),
                           PT := "pressure"."Over pressure Delay time user");
   "IEC_Timer_0_DB_9".TOF(IN := "IEC_Timer_0_DB_28".Q, PT := t#3s);
   "pressure"."Control A"."Over pressure occured" := "IEC_Timer_0_DB_9".Q;
END_REGION

REGION Network 11: gear pump B Over pressure
   RUNG wire#powerrail
      { S7_Templates := "SrcType := Real" } GT_Contact(in1 := "pressure"."pump B Inlet", in2 := "pressure"."B"."Maximum Pressure user")
      wire#w1
      { S7_Templates := "time_type := Time" } "IEC_Timer_0_DB_30".TON(pt := "pressure"."Over pressure Delay time user", et =>)
   END_RUNG
   RUNG wire#powerrail
      { S7_Templates := "SrcType := Real" } GT_Contact(in1 := "pressure"."pump B Inlet", in2 := "pressure"."B"."maximum pressure Admin")
   END_RUNG wire#w1
   RUNG wire#powerrail
      Contact( "IEC_Timer_0_DB_30".Q )
      { S7_Templates := "time_type := Time" } "IEC_Timer_0_DB_14".TOF(pt := t#3s, et =>)
      Coil( "pressure"."Control B"."Over pressure occured" )
   END_RUNG
   // the same network as SCL:
   "IEC_Timer_0_DB_30".TON(IN := ("pressure"."pump B Inlet" > "pressure"."B"."Maximum Pressure user") OR ("pressure"."pump B Inlet" > "pressure"."B"."maximum pressure Admin"),
                           PT := "pressure"."Over pressure Delay time user");
   "IEC_Timer_0_DB_14".TOF(IN := "IEC_Timer_0_DB_30".Q, PT := t#3s);
   "pressure"."Control B"."Over pressure occured" := "IEC_Timer_0_DB_14".Q;
END_REGION

REGION Network 12: gear pump A Under pressure
   RUNG wire#powerrail
      { S7_Templates := "SrcType := Real" } LT_Contact(in1 := "pressure"."pump A Inlet", in2 := "pressure"."A"."minimum Pressure")
      Contact( "Gear Pump A On_FWD" )
      { S7_Templates := "time_type := Time" } "IEC_Timer_0_DB_31".TON(pt := "pressure"."under pressure delay time", et =>)
      { S7_Templates := "time_type := Time" } "IEC_Timer_0_DB_39".TOF(pt := T#5S, et =>)
      wire#w1
      Coil( "pressure"."Control A"."under pressure Occured" )
   END_RUNG
   RUNG wire#w1
      Coil( "Alarm_DB".input.alarm[43] )
   END_RUNG
   // the same network as SCL:
   "IEC_Timer_0_DB_31".TON(IN := ("pressure"."pump A Inlet" < "pressure"."A"."minimum Pressure") AND "Gear Pump A On_FWD",
                           PT := "pressure"."under pressure delay time");
   "IEC_Timer_0_DB_39".TOF(IN := "IEC_Timer_0_DB_31".Q, PT := T#5S);
   "pressure"."Control A"."under pressure Occured" := "IEC_Timer_0_DB_39".Q;
   "Alarm_DB".input.alarm[43] := "IEC_Timer_0_DB_39".Q;
END_REGION

REGION Network 13: gear pump B under pressure
   RUNG wire#powerrail
      { S7_Templates := "SrcType := Real" } LT_Contact(in1 := "pressure"."pump B Inlet", in2 := "pressure"."B"."minimum Pressure")
      Contact( "Gear Pump B On_FWD" )
      { S7_Templates := "time_type := Time" } "IEC_Timer_0_DB_32".TON(pt := "pressure"."under pressure delay time", et =>)
      { S7_Templates := "time_type := Time" } "IEC_Timer_0_DB_40".TOF(pt := T#5S, et =>)
      wire#w1
      Coil( "pressure"."Control B"."under pressure Occured" )
   END_RUNG
   RUNG wire#w1
      Coil( "Alarm_DB".input.alarm[44] )
   END_RUNG
   // the same network as SCL:
   "IEC_Timer_0_DB_32".TON(IN := ("pressure"."pump B Inlet" < "pressure"."B"."minimum Pressure") AND "Gear Pump B On_FWD",
                           PT := "pressure"."under pressure delay time");
   "IEC_Timer_0_DB_40".TOF(IN := "IEC_Timer_0_DB_32".Q, PT := T#5S);
   "pressure"."Control B"."under pressure Occured" := "IEC_Timer_0_DB_40".Q;
   "Alarm_DB".input.alarm[44] := "IEC_Timer_0_DB_40".Q;
END_REGION

REGION Network 14: gear pump A Over pressure outlet
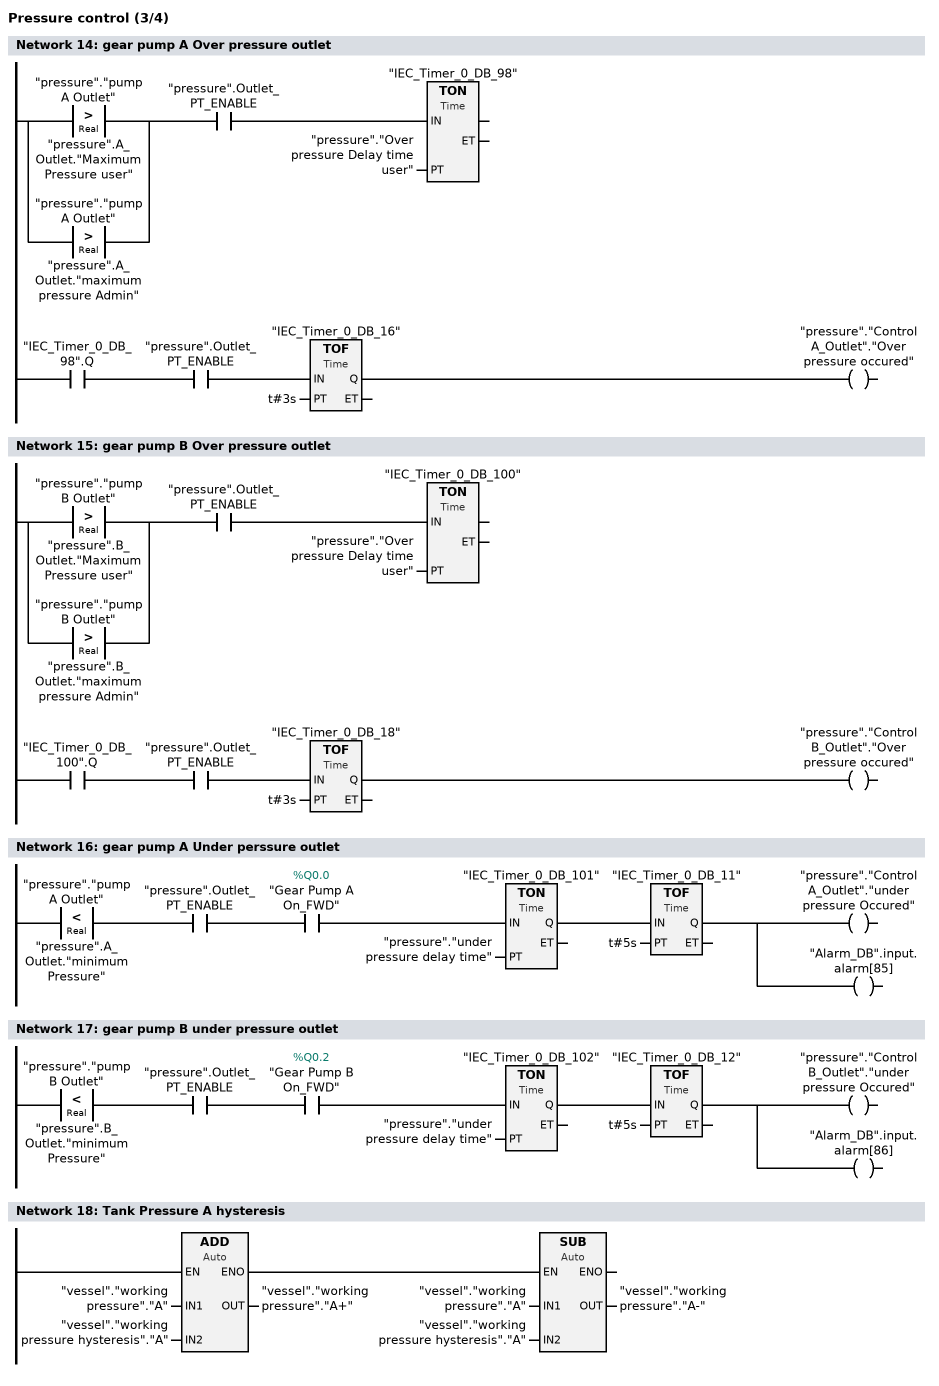
   RUNG wire#powerrail
      { S7_Templates := "SrcType := Real" } GT_Contact(in1 := "pressure"."pump A Outlet", in2 := "pressure".A_Outlet."Maximum Pressure user")
      wire#w1
      Contact( "pressure".Outlet_PT_ENABLE )
      { S7_Templates := "time_type := Time" } "IEC_Timer_0_DB_98".TON(pt := "pressure"."Over pressure Delay time user", et =>)
   END_RUNG
   RUNG wire#powerrail
      { S7_Templates := "SrcType := Real" } GT_Contact(in1 := "pressure"."pump A Outlet", in2 := "pressure".A_Outlet."maximum pressure Admin")
   END_RUNG wire#w1
   RUNG wire#powerrail
      Contact( "IEC_Timer_0_DB_98".Q )
      Contact( "pressure".Outlet_PT_ENABLE )
      { S7_Templates := "time_type := Time" } "IEC_Timer_0_DB_16".TOF(pt := t#3s, et =>)
      Coil( "pressure"."Control A_Outlet"."Over pressure occured" )
   END_RUNG
   // the same network as SCL:
   "IEC_Timer_0_DB_98".TON(IN := (("pressure"."pump A Outlet" > "pressure".A_Outlet."Maximum Pressure user") OR ("pressure"."pump A Outlet" > "pressure".A_Outlet."maximum pressure Admin")) AND "pressure".Outlet_PT_ENABLE,
                           PT := "pressure"."Over pressure Delay time user");
   "IEC_Timer_0_DB_16".TOF(IN := "IEC_Timer_0_DB_98".Q AND "pressure".Outlet_PT_ENABLE, PT := t#3s);
   "pressure"."Control A_Outlet"."Over pressure occured" := "IEC_Timer_0_DB_16".Q;
END_REGION

REGION Network 15: gear pump B Over pressure outlet
   RUNG wire#powerrail
      { S7_Templates := "SrcType := Real" } GT_Contact(in1 := "pressure"."pump B Outlet", in2 := "pressure".B_Outlet."Maximum Pressure user")
      wire#w1
      Contact( "pressure".Outlet_PT_ENABLE )
      { S7_Templates := "time_type := Time" } "IEC_Timer_0_DB_100".TON(pt := "pressure"."Over pressure Delay time user", et =>)
   END_RUNG
   RUNG wire#powerrail
      { S7_Templates := "SrcType := Real" } GT_Contact(in1 := "pressure"."pump B Outlet", in2 := "pressure".B_Outlet."maximum pressure Admin")
   END_RUNG wire#w1
   RUNG wire#powerrail
      Contact( "IEC_Timer_0_DB_100".Q )
      Contact( "pressure".Outlet_PT_ENABLE )
      { S7_Templates := "time_type := Time" } "IEC_Timer_0_DB_18".TOF(pt := t#3s, et =>)
      Coil( "pressure"."Control B_Outlet"."Over pressure occured" )
   END_RUNG
   // the same network as SCL:
   "IEC_Timer_0_DB_100".TON(IN := (("pressure"."pump B Outlet" > "pressure".B_Outlet."Maximum Pressure user") OR ("pressure"."pump B Outlet" > "pressure".B_Outlet."maximum pressure Admin")) AND "pressure".Outlet_PT_ENABLE,
                           PT := "pressure"."Over pressure Delay time user");
   "IEC_Timer_0_DB_18".TOF(IN := "IEC_Timer_0_DB_100".Q AND "pressure".Outlet_PT_ENABLE, PT := t#3s);
   "pressure"."Control B_Outlet"."Over pressure occured" := "IEC_Timer_0_DB_18".Q;
END_REGION

REGION Network 16: gear pump A Under perssure outlet
   RUNG wire#powerrail
      { S7_Templates := "SrcType := Real" } LT_Contact(in1 := "pressure"."pump A Outlet", in2 := "pressure".A_Outlet."minimum Pressure")
      Contact( "pressure".Outlet_PT_ENABLE )
      Contact( "Gear Pump A On_FWD" )
      { S7_Templates := "time_type := Time" } "IEC_Timer_0_DB_101".TON(pt := "pressure"."under pressure delay time", et =>)
      { S7_Templates := "time_type := Time" } "IEC_Timer_0_DB_11".TOF(pt := t#5s, et =>)
      wire#w1
      Coil( "pressure"."Control A_Outlet"."under pressure Occured" )
   END_RUNG
   RUNG wire#w1
      Coil( "Alarm_DB".input.alarm[85] )
   END_RUNG
   // the same network as SCL:
   "IEC_Timer_0_DB_101".TON(IN := ("pressure"."pump A Outlet" < "pressure".A_Outlet."minimum Pressure") AND "pressure".Outlet_PT_ENABLE AND "Gear Pump A On_FWD",
                           PT := "pressure"."under pressure delay time");
   "IEC_Timer_0_DB_11".TOF(IN := "IEC_Timer_0_DB_101".Q, PT := t#5s);
   "pressure"."Control A_Outlet"."under pressure Occured" := "IEC_Timer_0_DB_11".Q;
   "Alarm_DB".input.alarm[85] := "IEC_Timer_0_DB_11".Q;
END_REGION

REGION Network 17: gear pump B under pressure outlet
   RUNG wire#powerrail
      { S7_Templates := "SrcType := Real" } LT_Contact(in1 := "pressure"."pump B Outlet", in2 := "pressure".B_Outlet."minimum Pressure")
      Contact( "pressure".Outlet_PT_ENABLE )
      Contact( "Gear Pump B On_FWD" )
      { S7_Templates := "time_type := Time" } "IEC_Timer_0_DB_102".TON(pt := "pressure"."under pressure delay time", et =>)
      { S7_Templates := "time_type := Time" } "IEC_Timer_0_DB_12".TOF(pt := t#5s, et =>)
      wire#w1
      Coil( "pressure"."Control B_Outlet"."under pressure Occured" )
   END_RUNG
   RUNG wire#w1
      Coil( "Alarm_DB".input.alarm[86] )
   END_RUNG
   // the same network as SCL:
   "IEC_Timer_0_DB_102".TON(IN := ("pressure"."pump B Outlet" < "pressure".B_Outlet."minimum Pressure") AND "pressure".Outlet_PT_ENABLE AND "Gear Pump B On_FWD",
                           PT := "pressure"."under pressure delay time");
   "IEC_Timer_0_DB_12".TOF(IN := "IEC_Timer_0_DB_102".Q, PT := t#5s);
   "pressure"."Control B_Outlet"."under pressure Occured" := "IEC_Timer_0_DB_12".Q;
   "Alarm_DB".input.alarm[86] := "IEC_Timer_0_DB_12".Q;
END_REGION

REGION Network 18: Tank Pressure A hysteresis
   RUNG wire#powerrail
      Add(in1 := "vessel"."working pressure"."A", in2 := "vessel"."working pressure hysteresis"."A", out => "vessel"."working pressure"."A+")
      Sub(in1 := "vessel"."working pressure"."A", in2 := "vessel"."working pressure hysteresis"."A", out => "vessel"."working pressure"."A-")
   END_RUNG
   // the same network as SCL:
   "vessel"."working pressure"."A+" := "vessel"."working pressure"."A" + "vessel"."working pressure hysteresis"."A";
   "vessel"."working pressure"."A-" := "vessel"."working pressure"."A" - "vessel"."working pressure hysteresis"."A";
END_REGION

REGION Network 19: Tank Pressure B hysteresis
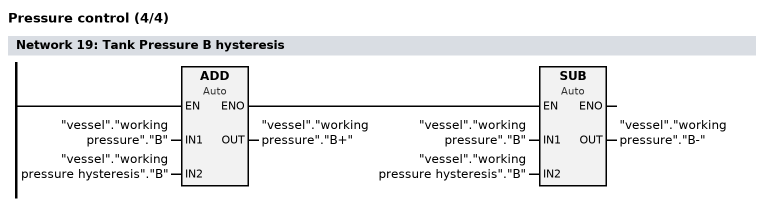
   RUNG wire#powerrail
      Add(in1 := "vessel"."working pressure"."B", in2 := "vessel"."working pressure hysteresis"."B", out => "vessel"."working pressure"."B+")
      Sub(in1 := "vessel"."working pressure"."B", in2 := "vessel"."working pressure hysteresis"."B", out => "vessel"."working pressure"."B-")
   END_RUNG
   // the same network as SCL:
   "vessel"."working pressure"."B+" := "vessel"."working pressure"."B" + "vessel"."working pressure hysteresis"."B";
   "vessel"."working pressure"."B-" := "vessel"."working pressure"."B" - "vessel"."working pressure hysteresis"."B";
END_REGION
END_FUNCTION

FUNCTION "Controls" : Void   // FC8, LAD
{ S7_Optimized_Access := 'TRUE' }
VERSION : 0.1
// stored: AutoNumber true, IsIECCheckEnabled false, SetENOAutomatically false, UDAEnableTagReadback false
BEGIN

REGION Network 1: Function selected
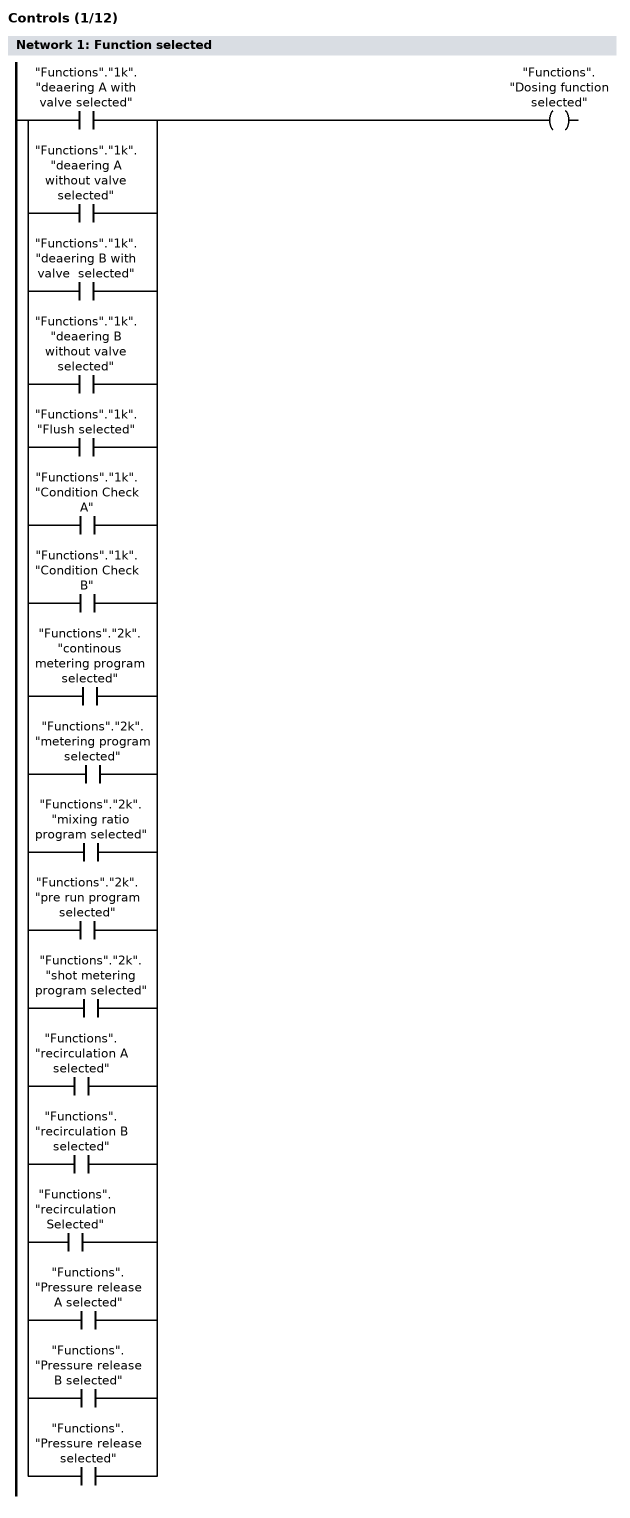
   RUNG wire#powerrail
      Contact( "Functions"."1k"."deaering A with valve selected" )
      wire#w1
      Coil( "Functions"."Dosing function selected" )
   END_RUNG
   RUNG wire#powerrail
      Contact( "Functions"."1k"."deaering A without valve selected" )
   END_RUNG wire#w1
   RUNG wire#powerrail
      Contact( "Functions"."1k"."deaering B with valve  selected" )
   END_RUNG wire#w1
   RUNG wire#powerrail
      Contact( "Functions"."1k"."deaering B without valve  selected" )
   END_RUNG wire#w1
   RUNG wire#powerrail
      Contact( "Functions"."1k"."Flush selected" )
   END_RUNG wire#w1
   RUNG wire#powerrail
      Contact( "Functions"."1k"."Condition Check A" )
   END_RUNG wire#w1
   RUNG wire#powerrail
      Contact( "Functions"."1k"."Condition Check B" )
   END_RUNG wire#w1
   RUNG wire#powerrail
      Contact( "Functions"."2k"."continous metering program selected" )
   END_RUNG wire#w1
   RUNG wire#powerrail
      Contact( "Functions"."2k"."metering program selected" )
   END_RUNG wire#w1
   RUNG wire#powerrail
      Contact( "Functions"."2k"."mixing ratio program selected" )
   END_RUNG wire#w1
   RUNG wire#powerrail
      Contact( "Functions"."2k"."pre run program selected" )
   END_RUNG wire#w1
   RUNG wire#powerrail
      Contact( "Functions"."2k"."shot metering program selected" )
   END_RUNG wire#w1
   RUNG wire#powerrail
      Contact( "Functions"."recirculation A selected" )
   END_RUNG wire#w1
   RUNG wire#powerrail
      Contact( "Functions"."recirculation B selected" )
   END_RUNG wire#w1
   RUNG wire#powerrail
      Contact( "Functions"."recirculation Selected" )
   END_RUNG wire#w1
   RUNG wire#powerrail
      Contact( "Functions"."Pressure release A selected" )
   END_RUNG wire#w1
   RUNG wire#powerrail
      Contact( "Functions"."Pressure release B selected" )
   END_RUNG wire#w1
   RUNG wire#powerrail
      Contact( "Functions"."Pressure release selected" )
   END_RUNG wire#w1
   // the same network as SCL:
   "Functions"."Dosing function selected" := "Functions"."1k"."deaering A with valve selected" OR "Functions"."1k"."deaering A without valve selected" OR "Functions"."1k"."deaering B with valve  selected" OR "Functions"."1k"."deaering B without valve  selected" OR "Functions"."1k"."Flush selected" OR "Functions"."1k"."Condition Check A" OR "Functions"."1k"."Condition Check B" OR "Functions"."2k"."continous metering program selected" OR "Functions"."2k"."metering program selected" OR "Functions"."2k"."mixing ratio program selected" OR "Functions"."2k"."pre run program selected" OR "Functions"."2k"."shot metering program selected" OR "Functions"."recirculation A selected" OR "Functions"."recirculation B selected" OR "Functions"."recirculation Selected" OR "Functions"."Pressure release A selected" OR "Functions"."Pressure release B selected" OR "Functions"."Pressure release selected";
END_REGION

REGION Network 2: Deselect all function
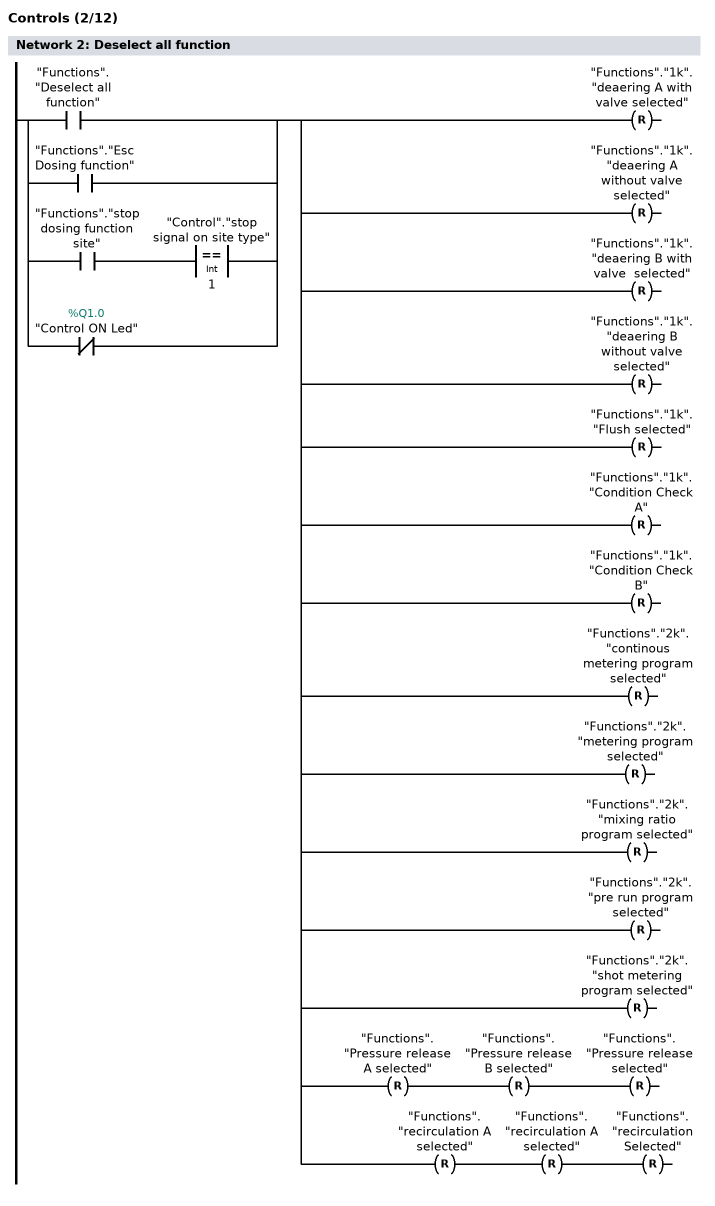
   RUNG wire#powerrail
      Contact( "Functions"."Deselect all function" )
      wire#w1
      R_Coil( "Functions"."1k"."deaering A with valve selected" )
   END_RUNG
   RUNG wire#powerrail
      Contact( "Functions"."Esc Dosing function" )
   END_RUNG wire#w1
   RUNG wire#powerrail
      Contact( "Functions"."stop dosing function site" )
      { S7_Templates := "SrcType := Int" } EQ_Contact(in1 := "Control"."stop signal on site type", in2 := 1)
   END_RUNG wire#w1
   RUNG wire#powerrail
      I_Contact( "Control ON Led" )
   END_RUNG wire#w1
   RUNG wire#w1
      R_Coil( "Functions"."1k"."deaering A without valve selected" )
   END_RUNG
   RUNG wire#w1
      R_Coil( "Functions"."1k"."deaering B with valve  selected" )
   END_RUNG
   RUNG wire#w1
      R_Coil( "Functions"."1k"."deaering B without valve  selected" )
   END_RUNG
   RUNG wire#w1
      R_Coil( "Functions"."1k"."Flush selected" )
   END_RUNG
   RUNG wire#w1
      R_Coil( "Functions"."1k"."Condition Check A" )
   END_RUNG
   RUNG wire#w1
      R_Coil( "Functions"."1k"."Condition Check B" )
   END_RUNG
   RUNG wire#w1
      R_Coil( "Functions"."2k"."continous metering program selected" )
   END_RUNG
   RUNG wire#w1
      R_Coil( "Functions"."2k"."metering program selected" )
   END_RUNG
   RUNG wire#w1
      R_Coil( "Functions"."2k"."mixing ratio program selected" )
   END_RUNG
   RUNG wire#w1
      R_Coil( "Functions"."2k"."pre run program selected" )
   END_RUNG
   RUNG wire#w1
      R_Coil( "Functions"."2k"."shot metering program selected" )
   END_RUNG
   RUNG wire#w1
      R_Coil( "Functions"."Pressure release A selected" )
      R_Coil( "Functions"."Pressure release B selected" )
      R_Coil( "Functions"."Pressure release selected" )
   END_RUNG
   RUNG wire#w1
      R_Coil( "Functions"."recirculation A selected" )
      R_Coil( "Functions"."recirculation A selected" )
      R_Coil( "Functions"."recirculation Selected" )
   END_RUNG
   // the same network as SCL:
   IF "Functions"."Deselect all function" OR "Functions"."Esc Dosing function" OR ("Functions"."stop dosing function site" AND ("Control"."stop signal on site type" = 1)) OR NOT "Control ON Led" THEN
       "Functions"."1k"."deaering A with valve selected" := FALSE;
       "Functions"."1k"."deaering A without valve selected" := FALSE;
       "Functions"."1k"."deaering B with valve  selected" := FALSE;
       "Functions"."1k"."deaering B without valve  selected" := FALSE;
       "Functions"."1k"."Flush selected" := FALSE;
       "Functions"."1k"."Condition Check A" := FALSE;
       "Functions"."1k"."Condition Check B" := FALSE;
       "Functions"."2k"."continous metering program selected" := FALSE;
       "Functions"."2k"."metering program selected" := FALSE;
       "Functions"."2k"."mixing ratio program selected" := FALSE;
       "Functions"."2k"."pre run program selected" := FALSE;
       "Functions"."2k"."shot metering program selected" := FALSE;
       "Functions"."Pressure release A selected" := FALSE;
       "Functions"."Pressure release B selected" := FALSE;
       "Functions"."Pressure release selected" := FALSE;
       "Functions"."recirculation A selected" := FALSE;
       "Functions"."recirculation A selected" := FALSE;
       "Functions"."recirculation Selected" := FALSE;
   END_IF;
END_REGION

REGION Network 3: Deselect all function During Refilling
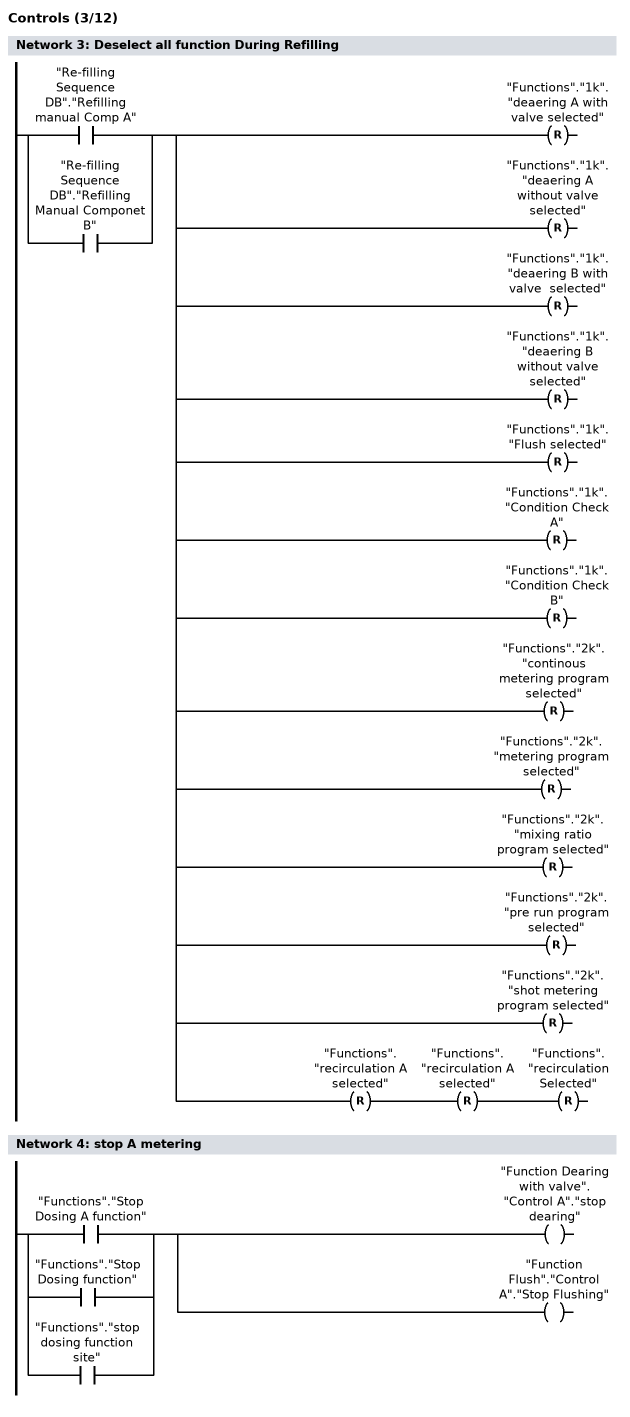
   RUNG wire#powerrail
      Contact( "Re-filling Sequence DB"."Refilling manual Comp A" )
      wire#w1
      R_Coil( "Functions"."1k"."deaering A with valve selected" )
   END_RUNG
   RUNG wire#powerrail
      Contact( "Re-filling Sequence DB"."Refilling Manual Componet B" )
   END_RUNG wire#w1
   RUNG wire#w1
      R_Coil( "Functions"."1k"."deaering A without valve selected" )
   END_RUNG
   RUNG wire#w1
      R_Coil( "Functions"."1k"."deaering B with valve  selected" )
   END_RUNG
   RUNG wire#w1
      R_Coil( "Functions"."1k"."deaering B without valve  selected" )
   END_RUNG
   RUNG wire#w1
      R_Coil( "Functions"."1k"."Flush selected" )
   END_RUNG
   RUNG wire#w1
      R_Coil( "Functions"."1k"."Condition Check A" )
   END_RUNG
   RUNG wire#w1
      R_Coil( "Functions"."1k"."Condition Check B" )
   END_RUNG
   RUNG wire#w1
      R_Coil( "Functions"."2k"."continous metering program selected" )
   END_RUNG
   RUNG wire#w1
      R_Coil( "Functions"."2k"."metering program selected" )
   END_RUNG
   RUNG wire#w1
      R_Coil( "Functions"."2k"."mixing ratio program selected" )
   END_RUNG
   RUNG wire#w1
      R_Coil( "Functions"."2k"."pre run program selected" )
   END_RUNG
   RUNG wire#w1
      R_Coil( "Functions"."2k"."shot metering program selected" )
   END_RUNG
   RUNG wire#w1
      R_Coil( "Functions"."recirculation A selected" )
      R_Coil( "Functions"."recirculation A selected" )
      R_Coil( "Functions"."recirculation Selected" )
   END_RUNG
   // the same network as SCL:
   IF "Re-filling Sequence DB"."Refilling manual Comp A" OR "Re-filling Sequence DB"."Refilling Manual Componet B" THEN
       "Functions"."1k"."deaering A with valve selected" := FALSE;
       "Functions"."1k"."deaering A without valve selected" := FALSE;
       "Functions"."1k"."deaering B with valve  selected" := FALSE;
       "Functions"."1k"."deaering B without valve  selected" := FALSE;
       "Functions"."1k"."Flush selected" := FALSE;
       "Functions"."1k"."Condition Check A" := FALSE;
       "Functions"."1k"."Condition Check B" := FALSE;
       "Functions"."2k"."continous metering program selected" := FALSE;
       "Functions"."2k"."metering program selected" := FALSE;
       "Functions"."2k"."mixing ratio program selected" := FALSE;
       "Functions"."2k"."pre run program selected" := FALSE;
       "Functions"."2k"."shot metering program selected" := FALSE;
       "Functions"."recirculation A selected" := FALSE;
       "Functions"."recirculation A selected" := FALSE;
       "Functions"."recirculation Selected" := FALSE;
   END_IF;
END_REGION

REGION Network 4: stop A metering
   RUNG wire#powerrail
      Contact( "Functions"."Stop Dosing A function" )
      wire#w1
      Coil( "Function Dearing with valve"."Control A"."stop dearing" )
   END_RUNG
   RUNG wire#powerrail
      Contact( "Functions"."Stop Dosing function" )
   END_RUNG wire#w1
   RUNG wire#powerrail
      Contact( "Functions"."stop dosing function site" )
   END_RUNG wire#w1
   RUNG wire#w1
      Coil( "Function Flush"."Control A"."Stop Flushing" )
   END_RUNG
   // the same network as SCL:
   "Function Dearing with valve"."Control A"."stop dearing" := "Functions"."Stop Dosing A function" OR "Functions"."Stop Dosing function" OR "Functions"."stop dosing function site";
   "Function Flush"."Control A"."Stop Flushing" := "Function Dearing with valve"."Control A"."stop dearing";
END_REGION

REGION Network 5: stop B metering
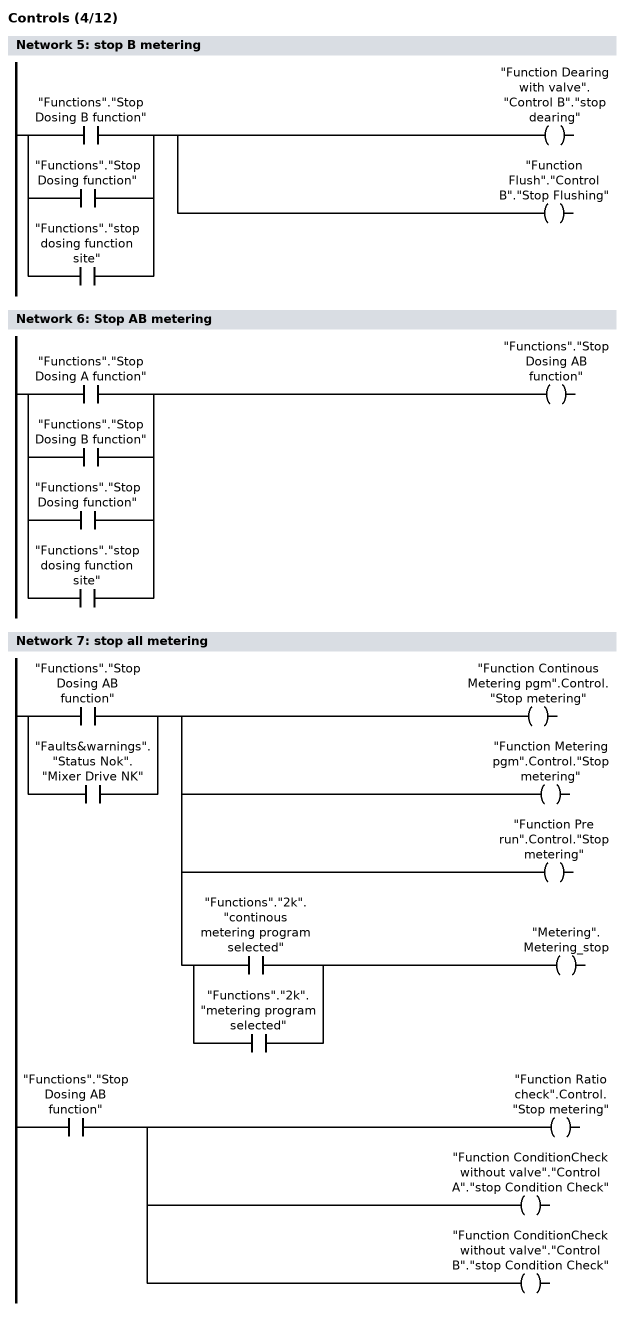
   RUNG wire#powerrail
      Contact( "Functions"."Stop Dosing B function" )
      wire#w1
      Coil( "Function Dearing with valve"."Control B"."stop dearing" )
   END_RUNG
   RUNG wire#powerrail
      Contact( "Functions"."Stop Dosing function" )
   END_RUNG wire#w1
   RUNG wire#powerrail
      Contact( "Functions"."stop dosing function site" )
   END_RUNG wire#w1
   RUNG wire#w1
      Coil( "Function Flush"."Control B"."Stop Flushing" )
   END_RUNG
   // the same network as SCL:
   "Function Dearing with valve"."Control B"."stop dearing" := "Functions"."Stop Dosing B function" OR "Functions"."Stop Dosing function" OR "Functions"."stop dosing function site";
   "Function Flush"."Control B"."Stop Flushing" := "Function Dearing with valve"."Control B"."stop dearing";
END_REGION

REGION Network 6: Stop AB metering
   RUNG wire#powerrail
      Contact( "Functions"."Stop Dosing A function" )
      wire#w1
      Coil( "Functions"."Stop Dosing AB function" )
   END_RUNG
   RUNG wire#powerrail
      Contact( "Functions"."Stop Dosing B function" )
   END_RUNG wire#w1
   RUNG wire#powerrail
      Contact( "Functions"."Stop Dosing function" )
   END_RUNG wire#w1
   RUNG wire#powerrail
      Contact( "Functions"."stop dosing function site" )
   END_RUNG wire#w1
   // the same network as SCL:
   "Functions"."Stop Dosing AB function" := "Functions"."Stop Dosing A function" OR "Functions"."Stop Dosing B function" OR "Functions"."Stop Dosing function" OR "Functions"."stop dosing function site";
END_REGION

REGION Network 7: stop all metering
   RUNG wire#powerrail
      Contact( "Functions"."Stop Dosing AB function" )
      wire#w1
      Coil( "Function Continous Metering pgm".Control."Stop metering" )
   END_RUNG
   RUNG wire#powerrail
      Contact( "Faults&warnings"."Status Nok"."Mixer Drive NK" )
   END_RUNG wire#w1
   RUNG wire#w1
      Coil( "Function Metering pgm".Control."Stop metering" )
   END_RUNG
   RUNG wire#w1
      Coil( "Function Pre run".Control."Stop metering" )
   END_RUNG
   RUNG wire#w1
      Contact( "Functions"."2k"."continous metering program selected" )
      wire#w2
      Coil( "Metering".Metering_stop )
   END_RUNG
   RUNG wire#w1
      Contact( "Functions"."2k"."metering program selected" )
   END_RUNG wire#w2
   RUNG wire#powerrail
      Contact( "Functions"."Stop Dosing AB function" )
      wire#w3
      Coil( "Function Ratio check".Control."Stop metering" )
   END_RUNG
   RUNG wire#w3
      Coil( "Function ConditionCheck without valve"."Control A"."stop Condition Check" )
   END_RUNG
   RUNG wire#w3
      Coil( "Function ConditionCheck without valve"."Control B"."stop Condition Check" )
   END_RUNG
   // the same network as SCL:
   "Function Continous Metering pgm".Control."Stop metering" := "Functions"."Stop Dosing AB function" OR "Faults&warnings"."Status Nok"."Mixer Drive NK";
   "Function Metering pgm".Control."Stop metering" := "Function Continous Metering pgm".Control."Stop metering";
   "Function Pre run".Control."Stop metering" := "Function Continous Metering pgm".Control."Stop metering";
   "Metering".Metering_stop := "Function Continous Metering pgm".Control."Stop metering" AND ("Functions"."2k"."continous metering program selected" OR "Functions"."2k"."metering program selected");
   "Function Ratio check".Control."Stop metering" := "Functions"."Stop Dosing AB function";
   "Function ConditionCheck without valve"."Control A"."stop Condition Check" := "Functions"."Stop Dosing AB function";
   "Function ConditionCheck without valve"."Control B"."stop Condition Check" := "Functions"."Stop Dosing AB function";
END_REGION

REGION Network 8: Critical fault Block A metering
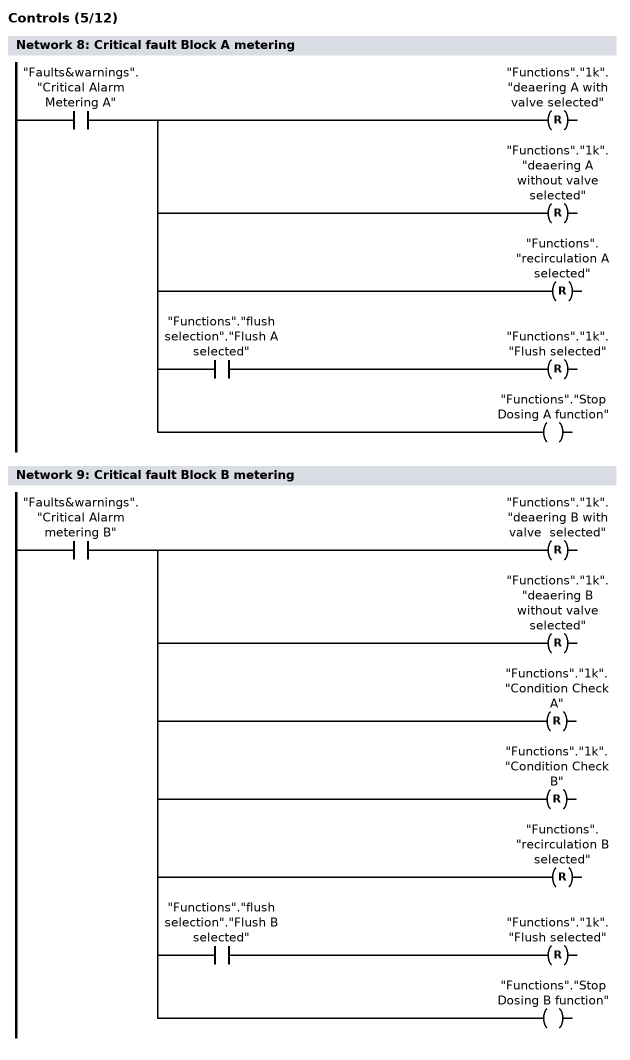
   RUNG wire#powerrail
      Contact( "Faults&warnings"."Critical Alarm Metering A" )
      wire#w1
      R_Coil( "Functions"."1k"."deaering A with valve selected" )
   END_RUNG
   RUNG wire#w1
      R_Coil( "Functions"."1k"."deaering A without valve selected" )
   END_RUNG
   RUNG wire#w1
      R_Coil( "Functions"."recirculation A selected" )
   END_RUNG
   RUNG wire#w1
      Contact( "Functions"."flush selection"."Flush A selected" )
      R_Coil( "Functions"."1k"."Flush selected" )
   END_RUNG
   RUNG wire#w1
      Coil( "Functions"."Stop Dosing A function" )
   END_RUNG
   // the same network as SCL:
   IF "Faults&warnings"."Critical Alarm Metering A" THEN
       "Functions"."1k"."deaering A with valve selected" := FALSE;
       "Functions"."1k"."deaering A without valve selected" := FALSE;
       "Functions"."recirculation A selected" := FALSE;
   END_IF;
   IF "Faults&warnings"."Critical Alarm Metering A" AND "Functions"."flush selection"."Flush A selected" THEN
       "Functions"."1k"."Flush selected" := FALSE;
   END_IF;
   "Functions"."Stop Dosing A function" := "Faults&warnings"."Critical Alarm Metering A";
END_REGION

REGION Network 9: Critical fault Block B metering
   RUNG wire#powerrail
      Contact( "Faults&warnings"."Critical Alarm metering B" )
      wire#w1
      R_Coil( "Functions"."1k"."deaering B with valve  selected" )
   END_RUNG
   RUNG wire#w1
      R_Coil( "Functions"."1k"."deaering B without valve  selected" )
   END_RUNG
   RUNG wire#w1
      R_Coil( "Functions"."1k"."Condition Check A" )
   END_RUNG
   RUNG wire#w1
      R_Coil( "Functions"."1k"."Condition Check B" )
   END_RUNG
   RUNG wire#w1
      R_Coil( "Functions"."recirculation B selected" )
   END_RUNG
   RUNG wire#w1
      Contact( "Functions"."flush selection"."Flush B selected" )
      R_Coil( "Functions"."1k"."Flush selected" )
   END_RUNG
   RUNG wire#w1
      Coil( "Functions"."Stop Dosing B function" )
   END_RUNG
   // the same network as SCL:
   IF "Faults&warnings"."Critical Alarm metering B" THEN
       "Functions"."1k"."deaering B with valve  selected" := FALSE;
       "Functions"."1k"."deaering B without valve  selected" := FALSE;
       "Functions"."1k"."Condition Check A" := FALSE;
       "Functions"."1k"."Condition Check B" := FALSE;
       "Functions"."recirculation B selected" := FALSE;
   END_IF;
   IF "Faults&warnings"."Critical Alarm metering B" AND "Functions"."flush selection"."Flush B selected" THEN
       "Functions"."1k"."Flush selected" := FALSE;
   END_IF;
   "Functions"."Stop Dosing B function" := "Faults&warnings"."Critical Alarm metering B";
END_REGION

REGION Network 10: Critical fault block all metering
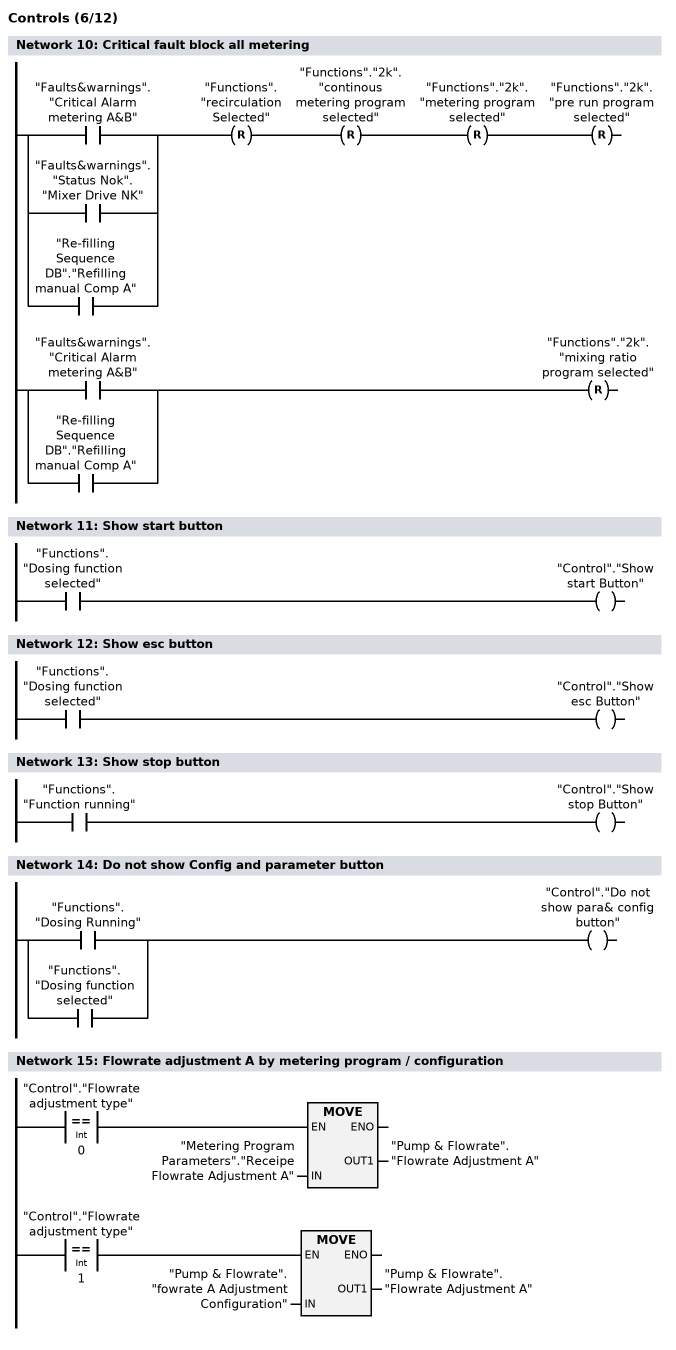
   RUNG wire#powerrail
      Contact( "Faults&warnings"."Critical Alarm metering A&B" )
      wire#w1
      R_Coil( "Functions"."recirculation Selected" )
      R_Coil( "Functions"."2k"."continous metering program selected" )
      R_Coil( "Functions"."2k"."metering program selected" )
      R_Coil( "Functions"."2k"."pre run program selected" )
   END_RUNG
   RUNG wire#powerrail
      Contact( "Faults&warnings"."Status Nok"."Mixer Drive NK" )
   END_RUNG wire#w1
   RUNG wire#powerrail
      Contact( "Re-filling Sequence DB"."Refilling manual Comp A" )
   END_RUNG wire#w1
   RUNG wire#powerrail
      Contact( "Faults&warnings"."Critical Alarm metering A&B" )
      wire#w2
      R_Coil( "Functions"."2k"."mixing ratio program selected" )
   END_RUNG
   RUNG wire#powerrail
      Contact( "Re-filling Sequence DB"."Refilling manual Comp A" )
   END_RUNG wire#w2
   // the same network as SCL:
   IF "Faults&warnings"."Critical Alarm metering A&B" OR "Faults&warnings"."Status Nok"."Mixer Drive NK" OR "Re-filling Sequence DB"."Refilling manual Comp A" THEN
       "Functions"."recirculation Selected" := FALSE;
       "Functions"."2k"."continous metering program selected" := FALSE;
       "Functions"."2k"."metering program selected" := FALSE;
       "Functions"."2k"."pre run program selected" := FALSE;
   END_IF;
   IF "Faults&warnings"."Critical Alarm metering A&B" OR "Re-filling Sequence DB"."Refilling manual Comp A" THEN
       "Functions"."2k"."mixing ratio program selected" := FALSE;
   END_IF;
END_REGION

REGION Network 11: Show start button
   RUNG wire#powerrail
      Contact( "Functions"."Dosing function selected" )
      Coil( "Control"."Show start Button" )
   END_RUNG
   // the same network as SCL:
   "Control"."Show start Button" := "Functions"."Dosing function selected";
END_REGION

REGION Network 12: Show esc button
   RUNG wire#powerrail
      Contact( "Functions"."Dosing function selected" )
      Coil( "Control"."Show esc Button" )
   END_RUNG
   // the same network as SCL:
   "Control"."Show esc Button" := "Functions"."Dosing function selected";
END_REGION

REGION Network 13: Show stop button
   RUNG wire#powerrail
      Contact( "Functions"."Function running" )
      Coil( "Control"."Show stop Button" )
   END_RUNG
   // the same network as SCL:
   "Control"."Show stop Button" := "Functions"."Function running";
END_REGION

REGION Network 14: Do not show Config and parameter button
   RUNG wire#powerrail
      Contact( "Functions"."Dosing Running" )
      wire#w1
      Coil( "Control"."Do not show para& config button" )
   END_RUNG
   RUNG wire#powerrail
      Contact( "Functions"."Dosing function selected" )
   END_RUNG wire#w1
   // the same network as SCL:
   "Control"."Do not show para& config button" := "Functions"."Dosing Running" OR "Functions"."Dosing function selected";
END_REGION

REGION Network 15: Flowrate adjustment A by metering program / configuration
   IF "Control"."Flowrate adjustment type" = 0 THEN
       "Pump & Flowrate"."Flowrate Adjustment A" := "Metering Program Parameters"."Receipe Flowrate Adjustment A";
   END_IF;
   IF "Control"."Flowrate adjustment type" = 1 THEN
       "Pump & Flowrate"."Flowrate Adjustment A" := "Pump & Flowrate"."fowrate A Adjustment Configuration";
   END_IF;
END_REGION

REGION Network 16: Flowrate adjustment B by metering program / configuration
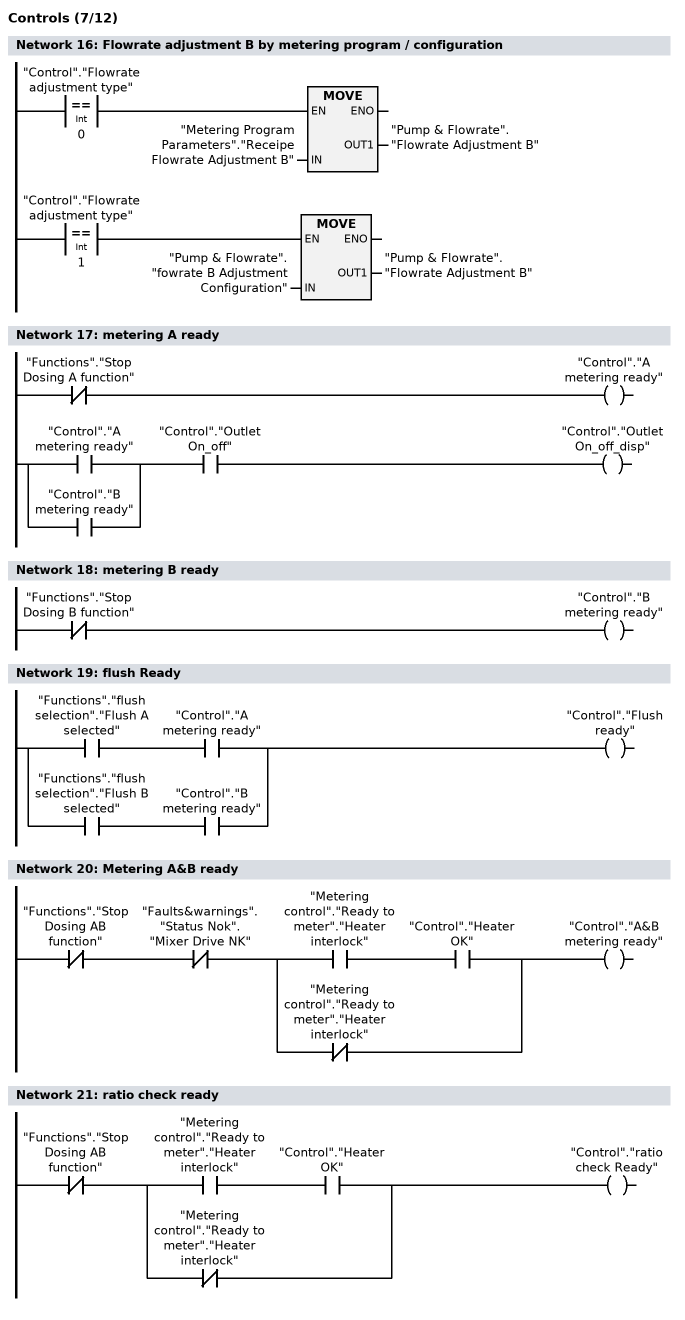
   IF "Control"."Flowrate adjustment type" = 0 THEN
       "Pump & Flowrate"."Flowrate Adjustment B" := "Metering Program Parameters"."Receipe Flowrate Adjustment B";
   END_IF;
   IF "Control"."Flowrate adjustment type" = 1 THEN
       "Pump & Flowrate"."Flowrate Adjustment B" := "Pump & Flowrate"."fowrate B Adjustment Configuration";
   END_IF;
END_REGION

REGION Network 17: metering A ready
   RUNG wire#powerrail
      I_Contact( "Functions"."Stop Dosing A function" )
      Coil( "Control"."A metering ready" )
   END_RUNG
   RUNG wire#powerrail
      Contact( "Control"."A metering ready" )
      wire#w1
      Contact( "Control"."Outlet On_off" )
      Coil( "Control"."Outlet On_off_disp" )
   END_RUNG
   RUNG wire#powerrail
      Contact( "Control"."B metering ready" )
   END_RUNG wire#w1
   // the same network as SCL:
   "Control"."A metering ready" := NOT "Functions"."Stop Dosing A function";
   "Control"."Outlet On_off_disp" := ("Control"."A metering ready" OR "Control"."B metering ready") AND "Control"."Outlet On_off";
END_REGION

REGION Network 18: metering B ready
   RUNG wire#powerrail
      I_Contact( "Functions"."Stop Dosing B function" )
      Coil( "Control"."B metering ready" )
   END_RUNG
   // the same network as SCL:
   "Control"."B metering ready" := NOT "Functions"."Stop Dosing B function";
END_REGION

REGION Network 19: flush Ready
   RUNG wire#powerrail
      Contact( "Functions"."flush selection"."Flush A selected" )
      Contact( "Control"."A metering ready" )
      wire#w1
      Coil( "Control"."Flush ready" )
   END_RUNG
   RUNG wire#powerrail
      Contact( "Functions"."flush selection"."Flush B selected" )
      Contact( "Control"."B metering ready" )
   END_RUNG wire#w1
   // the same network as SCL:
   "Control"."Flush ready" := ("Functions"."flush selection"."Flush A selected" AND "Control"."A metering ready") OR ("Functions"."flush selection"."Flush B selected" AND "Control"."B metering ready");
END_REGION

REGION Network 20: Metering A&B ready
   RUNG wire#powerrail
      I_Contact( "Functions"."Stop Dosing AB function" )
      I_Contact( "Faults&warnings"."Status Nok"."Mixer Drive NK" )
      wire#w1
      Contact( "Metering control"."Ready to meter"."Heater interlock" )
      Contact( "Control"."Heater OK" )
      wire#w2
      Coil( "Control"."A&B metering ready" )
   END_RUNG
   RUNG wire#w1
      I_Contact( "Metering control"."Ready to meter"."Heater interlock" )
   END_RUNG wire#w2
   // the same network as SCL:
   "Control"."A&B metering ready" := NOT "Functions"."Stop Dosing AB function" AND NOT "Faults&warnings"."Status Nok"."Mixer Drive NK" AND (("Metering control"."Ready to meter"."Heater interlock" AND "Control"."Heater OK") OR NOT "Metering control"."Ready to meter"."Heater interlock");
END_REGION

REGION Network 21: ratio check ready
   RUNG wire#powerrail
      I_Contact( "Functions"."Stop Dosing AB function" )
      wire#w1
      Contact( "Metering control"."Ready to meter"."Heater interlock" )
      Contact( "Control"."Heater OK" )
      wire#w2
      Coil( "Control"."ratio check Ready" )
   END_RUNG
   RUNG wire#w1
      I_Contact( "Metering control"."Ready to meter"."Heater interlock" )
   END_RUNG wire#w2
   // the same network as SCL:
   "Control"."ratio check Ready" := NOT "Functions"."Stop Dosing AB function" AND (("Metering control"."Ready to meter"."Heater interlock" AND "Control"."Heater OK") OR NOT "Metering control"."Ready to meter"."Heater interlock");
END_REGION

REGION Network 22: Metering program ready
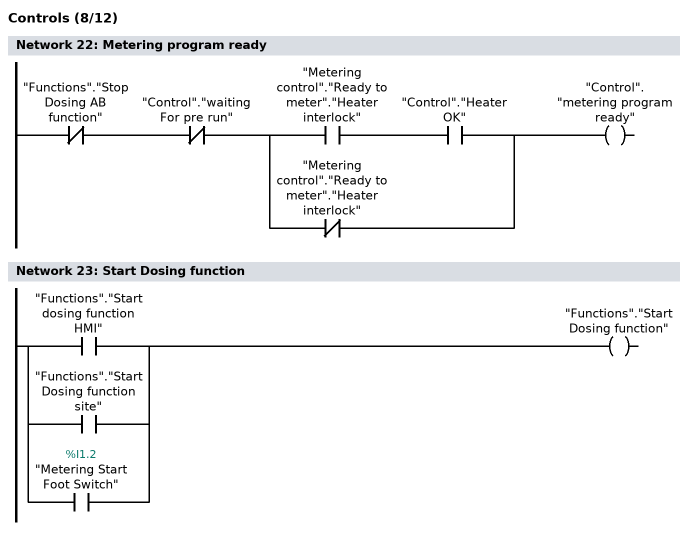
   RUNG wire#powerrail
      I_Contact( "Functions"."Stop Dosing AB function" )
      I_Contact( "Control"."waiting For pre run" )
      wire#w1
      Contact( "Metering control"."Ready to meter"."Heater interlock" )
      Contact( "Control"."Heater OK" )
      wire#w2
      Coil( "Control"."metering program ready" )
   END_RUNG
   RUNG wire#w1
      I_Contact( "Metering control"."Ready to meter"."Heater interlock" )
   END_RUNG wire#w2
   // the same network as SCL:
   "Control"."metering program ready" := NOT "Functions"."Stop Dosing AB function" AND NOT "Control"."waiting For pre run" AND (("Metering control"."Ready to meter"."Heater interlock" AND "Control"."Heater OK") OR NOT "Metering control"."Ready to meter"."Heater interlock");
END_REGION

REGION Network 23: Start Dosing function
   RUNG wire#powerrail
      Contact( "Functions"."Start dosing function HMI" )
      wire#w1
      Coil( "Functions"."Start Dosing function" )
   END_RUNG
   RUNG wire#powerrail
      Contact( "Functions"."Start Dosing function site" )
   END_RUNG wire#w1
   RUNG wire#powerrail
      Contact( "Metering Start Foot Switch" )
   END_RUNG wire#w1
   // the same network as SCL:
   "Functions"."Start Dosing function" := "Functions"."Start dosing function HMI" OR "Functions"."Start Dosing function site" OR "Metering Start Foot Switch";
END_REGION

REGION Network 24: Dosing running
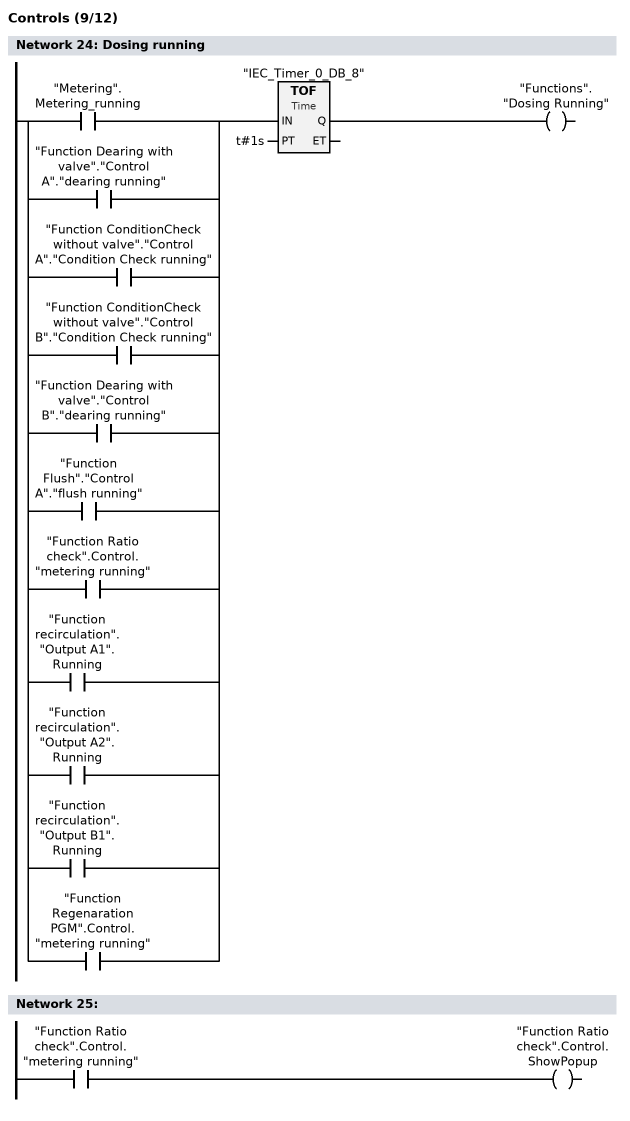
   RUNG wire#powerrail
      Contact( "Metering".Metering_running )
      wire#w1
      { S7_Templates := "time_type := Time" } "IEC_Timer_0_DB_8".TOF(pt := t#1s, et =>)
      Coil( "Functions"."Dosing Running" )
   END_RUNG
   RUNG wire#powerrail
      Contact( "Function Dearing with valve"."Control A"."dearing running" )
   END_RUNG wire#w1
   RUNG wire#powerrail
      Contact( "Function ConditionCheck without valve"."Control A"."Condition Check running" )
   END_RUNG wire#w1
   RUNG wire#powerrail
      Contact( "Function ConditionCheck without valve"."Control B"."Condition Check running" )
   END_RUNG wire#w1
   RUNG wire#powerrail
      Contact( "Function Dearing with valve"."Control B"."dearing running" )
   END_RUNG wire#w1
   RUNG wire#powerrail
      Contact( "Function Flush"."Control A"."flush running" )
   END_RUNG wire#w1
   RUNG wire#powerrail
      Contact( "Function Ratio check".Control."metering running" )
   END_RUNG wire#w1
   RUNG wire#powerrail
      Contact( "Function recirculation"."Output A1".Running )
   END_RUNG wire#w1
   RUNG wire#powerrail
      Contact( "Function recirculation"."Output A2".Running )
   END_RUNG wire#w1
   RUNG wire#powerrail
      Contact( "Function recirculation"."Output B1".Running )
   END_RUNG wire#w1
   RUNG wire#powerrail
      Contact( "Function Regenaration PGM".Control."metering running" )
   END_RUNG wire#w1
   // the same network as SCL:
   "IEC_Timer_0_DB_8".TOF(IN := "Metering".Metering_running OR "Function Dearing with valve"."Control A"."dearing running" OR "Function ConditionCheck without valve"."Control A"."Condition Check running" OR "Function ConditionCheck without valve"."Control B"."Condition Check running" OR "Function Dearing with valve"."Control B"."dearing running" OR "Function Flush"."Control A"."flush running" OR "Function Ratio check".Control."metering running" OR "Function recirculation"."Output A1".Running OR "Function recirculation"."Output A2".Running OR "Function recirculation"."Output B1".Running OR "Function Regenaration PGM".Control."metering running",
                          PT := t#1s);
   "Functions"."Dosing Running" := "IEC_Timer_0_DB_8".Q;
END_REGION

REGION Network 25
   RUNG wire#powerrail
      Contact( "Function Ratio check".Control."metering running" )
      Coil( "Function Ratio check".Control.ShowPopup )
   END_RUNG
   // the same network as SCL:
   "Function Ratio check".Control.ShowPopup := "Function Ratio check".Control."metering running";
END_REGION

REGION Network 26
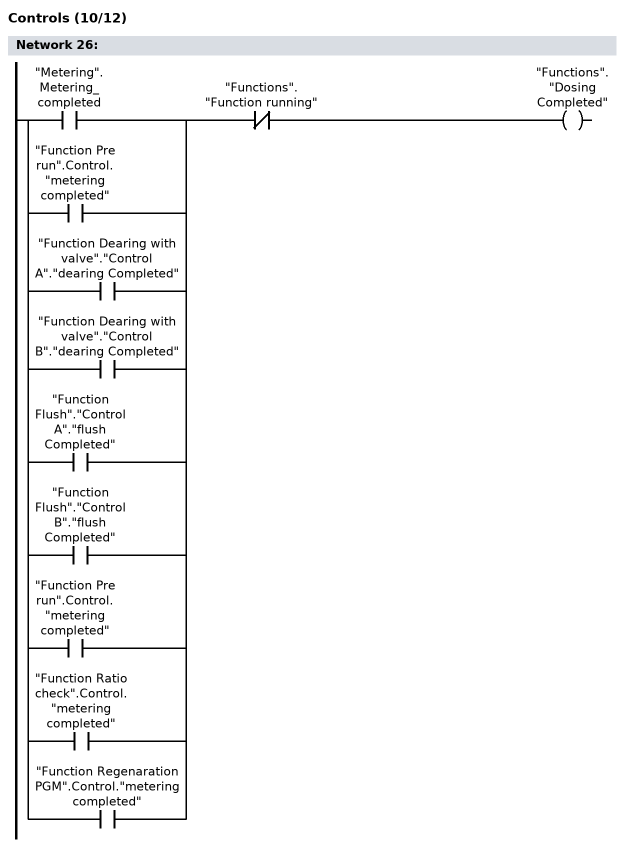
   RUNG wire#powerrail
      Contact( "Metering".Metering_completed )
      wire#w1
      I_Contact( "Functions"."Function running" )
      Coil( "Functions"."Dosing Completed" )
   END_RUNG
   RUNG wire#powerrail
      Contact( "Function Pre run".Control."metering completed" )
   END_RUNG wire#w1
   RUNG wire#powerrail
      Contact( "Function Dearing with valve"."Control A"."dearing Completed" )
   END_RUNG wire#w1
   RUNG wire#powerrail
      Contact( "Function Dearing with valve"."Control B"."dearing Completed" )
   END_RUNG wire#w1
   RUNG wire#powerrail
      Contact( "Function Flush"."Control A"."flush Completed" )
   END_RUNG wire#w1
   RUNG wire#powerrail
      Contact( "Function Flush"."Control B"."flush Completed" )
   END_RUNG wire#w1
   RUNG wire#powerrail
      Contact( "Function Pre run".Control."metering completed" )
   END_RUNG wire#w1
   RUNG wire#powerrail
      Contact( "Function Ratio check".Control."metering completed" )
   END_RUNG wire#w1
   RUNG wire#powerrail
      Contact( "Function Regenaration PGM".Control."metering completed" )
   END_RUNG wire#w1
   // the same network as SCL:
   "Functions"."Dosing Completed" := ("Metering".Metering_completed OR "Function Pre run".Control."metering completed" OR "Function Dearing with valve"."Control A"."dearing Completed" OR "Function Dearing with valve"."Control B"."dearing Completed" OR "Function Flush"."Control A"."flush Completed" OR "Function Flush"."Control B"."flush Completed" OR "Function Pre run".Control."metering completed" OR "Function Ratio check".Control."metering completed" OR "Function Regenaration PGM".Control."metering completed") AND NOT "Functions"."Function running";
END_REGION

REGION Network 27: Function running
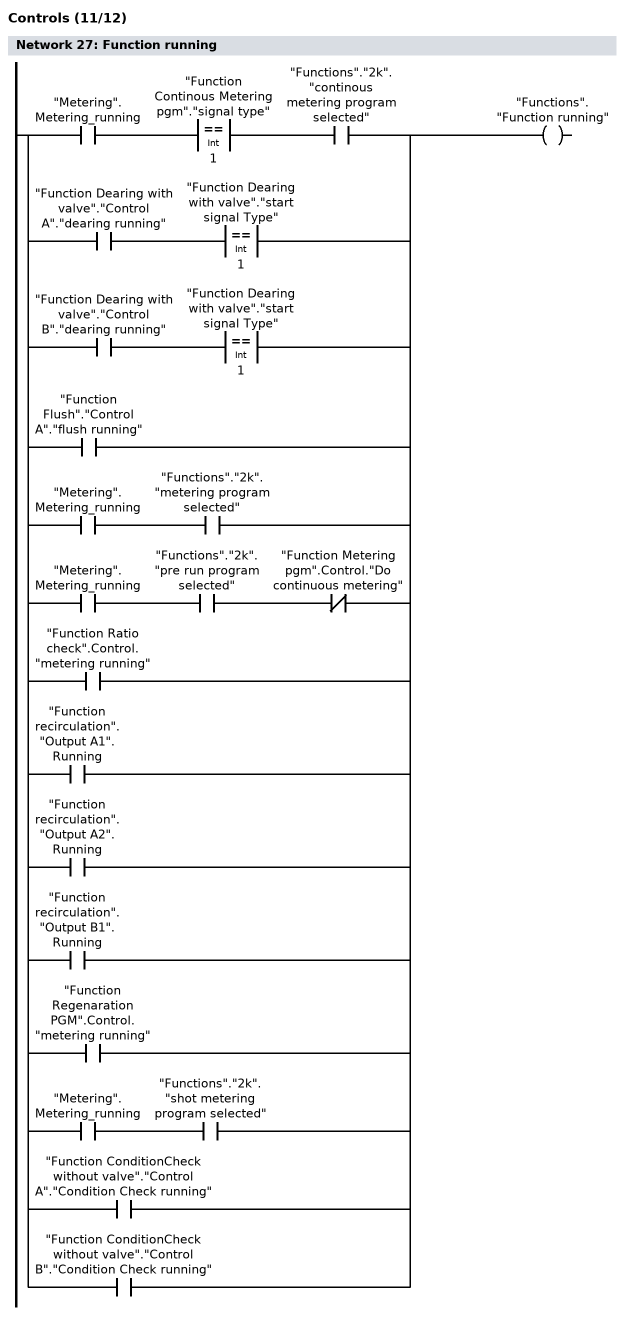
   RUNG wire#powerrail
      Contact( "Metering".Metering_running )
      { S7_Templates := "SrcType := Int" } EQ_Contact(in1 := "Function Continous Metering pgm"."signal type", in2 := 1)
      Contact( "Functions"."2k"."continous metering program selected" )
      wire#w1
      Coil( "Functions"."Function running" )
   END_RUNG
   RUNG wire#powerrail
      Contact( "Function Dearing with valve"."Control A"."dearing running" )
      { S7_Templates := "SrcType := Int" } EQ_Contact(in1 := "Function Dearing with valve"."start signal Type", in2 := 1)
   END_RUNG wire#w1
   RUNG wire#powerrail
      Contact( "Function Dearing with valve"."Control B"."dearing running" )
      { S7_Templates := "SrcType := Int" } EQ_Contact(in1 := "Function Dearing with valve"."start signal Type", in2 := 1)
   END_RUNG wire#w1
   RUNG wire#powerrail
      Contact( "Function Flush"."Control A"."flush running" )
   END_RUNG wire#w1
   RUNG wire#powerrail
      Contact( "Metering".Metering_running )
      Contact( "Functions"."2k"."metering program selected" )
   END_RUNG wire#w1
   RUNG wire#powerrail
      Contact( "Metering".Metering_running )
      Contact( "Functions"."2k"."pre run program selected" )
      I_Contact( "Function Metering pgm".Control."Do continuous metering" )
   END_RUNG wire#w1
   RUNG wire#powerrail
      Contact( "Function Ratio check".Control."metering running" )
   END_RUNG wire#w1
   RUNG wire#powerrail
      Contact( "Function recirculation"."Output A1".Running )
   END_RUNG wire#w1
   RUNG wire#powerrail
      Contact( "Function recirculation"."Output A2".Running )
   END_RUNG wire#w1
   RUNG wire#powerrail
      Contact( "Function recirculation"."Output B1".Running )
   END_RUNG wire#w1
   RUNG wire#powerrail
      Contact( "Function Regenaration PGM".Control."metering running" )
   END_RUNG wire#w1
   RUNG wire#powerrail
      Contact( "Metering".Metering_running )
      Contact( "Functions"."2k"."shot metering program selected" )
   END_RUNG wire#w1
   RUNG wire#powerrail
      Contact( "Function ConditionCheck without valve"."Control A"."Condition Check running" )
   END_RUNG wire#w1
   RUNG wire#powerrail
      Contact( "Function ConditionCheck without valve"."Control B"."Condition Check running" )
   END_RUNG wire#w1
   // the same network as SCL:
   "Functions"."Function running" := ("Metering".Metering_running AND ("Function Continous Metering pgm"."signal type" = 1) AND "Functions"."2k"."continous metering program selected") OR ("Function Dearing with valve"."Control A"."dearing running" AND ("Function Dearing with valve"."start signal Type" = 1)) OR ("Function Dearing with valve"."Control B"."dearing running" AND ("Function Dearing with valve"."start signal Type" = 1)) OR "Function Flush"."Control A"."flush running" OR ("Metering".Metering_running AND "Functions"."2k"."metering program selected") OR ("Metering".Metering_running AND "Functions"."2k"."pre run program selected" AND NOT "Function Metering pgm".Control."Do continuous metering") OR "Function Ratio check".Control."metering running" OR "Function recirculation"."Output A1".Running OR "Function recirculation"."Output A2".Running OR "Function recirculation"."Output B1".Running OR "Function Regenaration PGM".Control."metering running" OR ("Metering".Metering_running AND "Functions"."2k"."shot metering program selected") OR "Function ConditionCheck without valve"."Control A"."Condition Check running" OR "Function ConditionCheck without valve"."Control B"."Condition Check running";
END_REGION

REGION Network 28: show alarm textfield in all screen
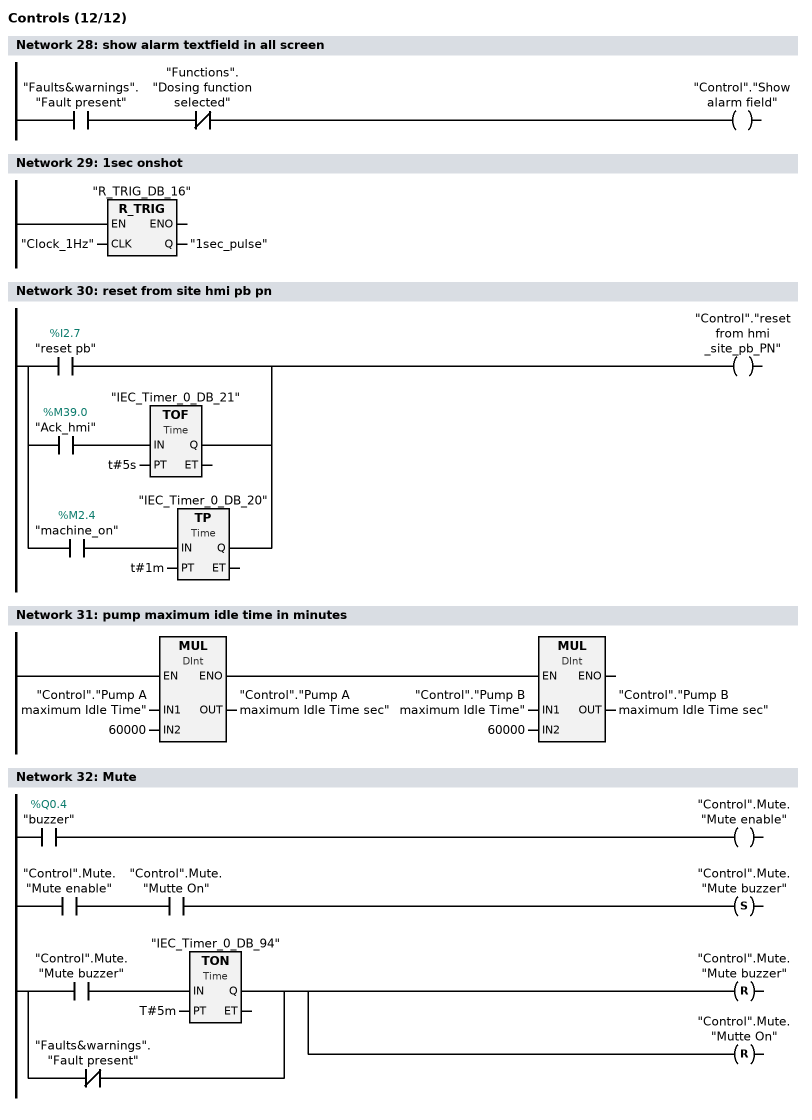
   RUNG wire#powerrail
      Contact( "Faults&warnings"."Fault present" )
      I_Contact( "Functions"."Dosing function selected" )
      Coil( "Control"."Show alarm field" )
   END_RUNG
   // the same network as SCL:
   "Control"."Show alarm field" := "Faults&warnings"."Fault present" AND NOT "Functions"."Dosing function selected";
END_REGION

REGION Network 29: 1sec onshot
   RUNG wire#powerrail
      "R_TRIG_DB_16".R_TRIG(CLK := "Clock_1Hz", Q => "1sec_pulse")
   END_RUNG
   // the same network as SCL:
   "R_TRIG_DB_16"(CLK := "Clock_1Hz", Q => "1sec_pulse");   // R_TRIG
END_REGION

REGION Network 30: reset from site hmi pb pn
   RUNG wire#powerrail
      Contact( "reset pb" )
      wire#w1
      Coil( "Control"."reset from hmi _site_pb_PN" )
   END_RUNG
   RUNG wire#powerrail
      Contact( "Ack_hmi" )
      { S7_Templates := "time_type := Time" } "IEC_Timer_0_DB_21".TOF(pt := t#5s, et =>)
   END_RUNG wire#w1
   RUNG wire#powerrail
      Contact( "machine_on" )
      { S7_Templates := "time_type := Time" } "IEC_Timer_0_DB_20".TP(pt := t#1m, et =>)
   END_RUNG wire#w1
   // the same network as SCL:
   "IEC_Timer_0_DB_21".TOF(IN := "Ack_hmi", PT := t#5s);
   "IEC_Timer_0_DB_20".TP(IN := "machine_on", PT := t#1m);
   "Control"."reset from hmi _site_pb_PN" := "reset pb" OR "IEC_Timer_0_DB_21".Q OR "IEC_Timer_0_DB_20".Q;
END_REGION

REGION Network 31: pump maximum idle time in minutes
   RUNG wire#powerrail
      { S7_Templates := "SrcType := DInt" } Mul(in1 := "Control"."Pump A maximum Idle Time", in2 := 60000, out => "Control"."Pump A maximum Idle Time sec")
      { S7_Templates := "SrcType := DInt" } Mul(in1 := "Control"."Pump B maximum Idle Time", in2 := 60000, out => "Control"."Pump B maximum Idle Time sec")
   END_RUNG
   // the same network as SCL:
   "Control"."Pump A maximum Idle Time sec" := "Control"."Pump A maximum Idle Time" * 60000;
   "Control"."Pump B maximum Idle Time sec" := "Control"."Pump B maximum Idle Time" * 60000;
END_REGION

REGION Network 32: Mute
   RUNG wire#powerrail
      Contact( "buzzer" )
      Coil( "Control".Mute."Mute enable" )
   END_RUNG
   RUNG wire#powerrail
      Contact( "Control".Mute."Mute enable" )
      Contact( "Control".Mute."Mutte On" )
      S_Coil( "Control".Mute."Mute buzzer" )
   END_RUNG
   RUNG wire#powerrail
      Contact( "Control".Mute."Mute buzzer" )
      { S7_Templates := "time_type := Time" } "IEC_Timer_0_DB_94".TON(pt := T#5m, et =>)
      wire#w1
      R_Coil( "Control".Mute."Mute buzzer" )
   END_RUNG
   RUNG wire#powerrail
      I_Contact( "Faults&warnings"."Fault present" )
   END_RUNG wire#w1
   RUNG wire#w1
      R_Coil( "Control".Mute."Mutte On" )
   END_RUNG
   // the same network as SCL:
   "Control".Mute."Mute enable" := "buzzer";
   IF "Control".Mute."Mute enable" AND "Control".Mute."Mutte On" THEN
       "Control".Mute."Mute buzzer" := TRUE;
   END_IF;
   "IEC_Timer_0_DB_94".TON(IN := "Control".Mute."Mute buzzer", PT := T#5m);
   IF "IEC_Timer_0_DB_94".Q OR NOT "Faults&warnings"."Fault present" THEN
       "Control".Mute."Mute buzzer" := FALSE;
       "Control".Mute."Mutte On" := FALSE;
   END_IF;
END_REGION
END_FUNCTION

FUNCTION "Pop-up Animation" : Void
{ S7_Optimized_Access := 'TRUE' }
VERSION : 0.1

BEGIN
	/// Additional Metering Pop-up enable
	
	
	//IF "HMI"."Current screen No" <> 1 THEN
	   // "Pop-up Db"."General Visibility" := 0;
	//END_IF;
	//& "HMI"."Current screen No"=1
	IF "Pop-up Db"."Additional metering Popup-enable" = 1  THEN
	    "Pop-up Db"."General Visibility" := 1;
	ELSE
	    "Pop-up Db"."General Visibility" := 0;
	    
	END_IF;
	// Pop-up Close
	IF "Pop-up Db"."Close Button" = 1 THEN
	    "Pop-up Db"."Additional metering Popup-enable" := 0;
	    "Pop-up Db"."General Visibility" := 0;
	    "Pop-up Db"."Close Button" := 0;
	    
	    "Pop-up Db"."Additional metering Popup-enable" := 0;
	END_IF;
	//Dearing A 
	IF "Control"."A metering ready" & "Pop-up Db"."Additional metering Popup-enable"= 1 THEN
	    "Pop-up Db"."Dearing A Visibility" := 1;
	ELSE
	    "Pop-up Db"."Dearing A Visibility" := 0;
	    
	  END_IF;
	  
	  IF "Control"."A metering ready" &  "pressure".Outlet_PT_ENABLE = 1 AND "Function ConditionCheck without valve".Condition_check_en THEN
	      //"Pop-up Db"."Additional metering Popup-enable" = 1 AND
	      "Pop-up Db"."Condition check visibility" := 1;
	      "Pop-up Db".parameter_scrno_condchecken := '10';
	  ELSE
	    "Pop-up Db"."Condition check visibility" := 0;
	    "Pop-up Db".parameter_scrno_condchecken := '09';
	  END_IF;
	//Re-circulation A
	//IF "Control"."A recirculation Ready" AND "Pop-up Db"."Additional metering Popup-enable"= 1 THEN
	    //"Pop-up Db"."Recirculation A Visibility" := 1;
	//ELSE
	    //"Pop-up Db"."Recirculation A Visibility" := 0;
	//END_IF;
	//Dearing B
	  IF "Control"."B metering ready" & "Pop-up Db"."Additional metering Popup-enable" = 1  THEN
	    "Pop-up Db"."Dearing B Visibility" := 1;
	ELSE
	    "Pop-up Db"."Dearing B Visibility" := 0;
	END_IF;
	//Dearing C
	///IF NOT "Functions"."Stop Dosing C function"  & "Pop-up Db"."Additional metering Popup-enable"= 1  THEN
	   /// "Pop-up Db"."Dearing C Visibility":=1;
	///ELSE
	   /// "Pop-up Db"."Dearing C Visibility" := 0;
	    
	///END_IF;
	
	
END_FUNCTION

FUNCTION "Function Selection HMI _Site_PB" : Void   // FC30, LAD
{ S7_Optimized_Access := 'TRUE' }
VERSION : 0.1
// stored: AutoNumber true, IsIECCheckEnabled false, SetENOAutomatically false, UDAEnableTagReadback false
   VAR_TEMP
      temp_unitsel : Int;
   END_VAR
   VAR_TEMP   // added for the SCL form of the ladder/FBD networks
      _w1 : Bool;
      _w2 : Bool;
   END_VAR
BEGIN

REGION Network 1: No functions selected
